	// instrument type
	g_instruIDs :ARRAY[1..g_instruTypesNum] OF INT :=[7, 8, 9, 10, 11, 12, 13, 14, 15, 16, 17, 20, 42, 43];
	
	// instrument name
	g_instruNullName :STRING := 'NULL';
	g_instruTotalLife : ARRAY[1..g_instruTypesNum] OF UINT := [11(20),100,1,1];
	g_instruNameString:ARRAY[1..g_instruTypesNum] OF STRING:=['Cadiere Forceps','Large Needle Driver','Mega SutureCut Needle Driver','Large SutureCut Needle Driver',	
															'RoundTip Scissors','Prograsp',	'Maryland Bipolar Forceps','Fenestrated Bipolar Forceps', 'Monopolar Curved Scissors',
															'Permanent Cautery Hook','Permanent Cautery Spatula','Camera','Ultrasonic Scalpel 45cm','Ultrasonic Scalpel 55cm'];
	//instrument chinese name
	g_instruNameStringCH:ARRAY[1..g_instruTypesNum] OF WSTRING:=["无创抓钳","持针钳","大号带剪刀持针钳","带剪刀持针钳","圆头直剪","细齿无创抓钳",
															"双极弧形电凝钳","双极鸭嘴电凝钳","单极弧剪","单极电钩", "单极电铲","内窥镜","超声刀 46cm","超声刀 55cm"];
	// instrument kinematic
	g_instruRodLength :ARRAY[1..g_instruTypesNum] OF LREAL :=[	0.5438,0.5438,0.5438,0.5438,	 0.5438,0.5438,0.5438, 0.5438,0.5438,	0.5432, 0.5432,0.49,0.46463,0.55225];
	g_instruHeadLength :ARRAY[1..g_instruTypesNum] OF LREAL :=[ 0.0089,0.0089,0.010,0.010,		 0.0089,0.01065,0.01065,0.01065,0.0091,	0.00935,0.00935, 0, 0, 0];
	g_instruFingerLength :ARRAY[1..g_instruTypesNum] OF LREAL :=[0.01950, 0.0096, 0.0109, 0.011, 0.01102, 0.02313, 0.019473, 0.0207, 0.01293, 0.01638, 0.01905, 0, 0, 0];

	k13:ARRAY[1..g_instruTypesNum] OF LREAL:=[0.775510204, 0.808510638, 0.590163934, 0.590163934,  0.791666667,  0.496732026, 0.590163934, 0.590163934, 0.75,   -0.663636364,	-0.663636364,   1, 1, 1];
	k23:ARRAY[1..g_instruTypesNum] OF LREAL:=[0.775510204,0.808510638, 0.590163934, 0.590163934,  0.791666667, 0.496732026, 0.590163934, 0.590163934,  0.75,   -0.663636364,	-0.663636364,   1, 1, 1];
	kx:ARRAY[1..g_instruTypesNum] OF LREAL:=[g_instruTypesNum(-1)];
	ky:ARRAY[1..g_instruTypesNum] OF LREAL:=[0.947368421, 0.947368421,0.947368421, 0.947368421, 0.947368421, 0.947368421, 0.947368421, 0.947368421, 0.947368421, 0.877192982, 0.877192982, 1, 1, 1];
	kz:ARRAY[1..g_instruTypesNum] OF LREAL:=[0.859649123, 0.824561404, 1.070175439, 1.070175439, 0.842105263, 1.342105263, 1.070175439, 1.070175439, 0.842105263, 0.964912281, 0.964912281, 1, 1, 1];
	
	g_instruMaxGripAngle:ARRAY[1..g_instruTypesNum] OF LREAL:=[45*g_deg2Rad, 40*g_deg2Rad, 40*g_deg2Rad, 40*g_deg2Rad, 40*g_deg2Rad, PI/2, 55*g_deg2Rad, 55*g_deg2Rad, PI/3, PI/6, PI/6,0,PI/4,PI/4];
	
	g_instruMaxRollAngle:ARRAY[1..g_instruTypesNum] OF LREAL:=[12(5.5), 2(g_largeNum)];
	g_instruMaxPitchAngle:ARRAY[1..g_instruTypesNum] OF LREAL:=[11(75*g_deg2Rad), 3(1)];
	g_instruMaxYawAngle:ARRAY[1..g_instruTypesNum] OF LREAL:=[9(PI/2), 90*g_deg2Rad, 90*g_deg2Rad, 3(1)];
	

	// master gripper angle limit
	g_maxMasterGripAngle :LREAL := 30*g_deg2Rad;
	g_minMasterGripAngle : LREAL :=0.0;
	g_masterGripForceStartAng :LREAL :=5*g_deg2Rad;
	
	//ultrasound knife kinematics parameter
	g_uknifeGripTravel :LREAL:= 0.00353;
	g_uknifeGripDividAngle : LREAL := 17 * g_deg2Rad;
	g_uknifeMotorLead : LREAL := 0.025;
	g_uknifeLeverRatio : LREAL := 13.0/18.5;
	
	// instrument backslash
	g_instruYawBacklash :ARRAY[1..g_instruTypesNum] OF LREAL :=[4.0*g_deg2rad, 4.0*g_deg2rad, 4.0*g_deg2rad, 4.0*g_deg2rad, 4.0*g_deg2rad, 4.0*g_deg2rad, 4.0*g_deg2rad, 4.0*g_deg2rad, 4.0*g_deg2rad,  8.0*g_deg2rad,  8.0*g_deg2rad,  0 , 0,  0 ];
	g_instruPitchBacklash :ARRAY[1..g_instruTypesNum] OF LREAL :=[3.0*g_deg2rad, 3.0*g_deg2rad, 3.0*g_deg2rad, 3.0*g_deg2rad, 3.0*g_deg2rad, 3.0*g_deg2rad, 3.0*g_deg2rad, 3.0*g_deg2rad, 3.0*g_deg2rad,  3.0*g_deg2rad,  3*g_deg2rad,  0 , 0,  0 ];
	g_instruBacklashDir: ARRAY[1..g_instruTypesNum] OF INT :=[-1, -1, -1, 0, 0];
	g_gripperCloseAng :LREAL := 2.0*g_deg2rad;
	
	// instrument grip yaw compensation
	g_instruGripYawCompAng :ARRAY[1..4] OF LREAL := [ 2*g_deg2rad,  4*g_deg2rad,  6*g_deg2rad,  8*g_deg2rad];
	g_instruGripYawCompForceLevel  :ARRAY[1..4] OF INT := [ 20, 40, 70, 101];
	
END_VAR

// ---- GVLs/GVL_interactUI.TcGVL
{attribute 'qualified_only'}
VAR_GLOBAL
	//read from UI
	//surgical status: true surgical start   false surgical finshed
	g_surgicalStatus : BOOL;

	//surgical site selection
	g_surgicalSite : UINT;

	//surgical location selection
	g_surgicalLocation : UINT;

	//stand column height limit : design 1805mm - 2495mm 
	g_heightLimit : UINT;
	g_heightLimitFromUI : UINT;
	g_heightLimitEnbale : BOOL;
	
	//ui control button enable
	g_uiCtrl : ST_uiControl;

	//ui send reset fault
	g_uiFaultReset : UINT;

	//write UI 
	//error code ID
	g_errIdType3 : UDINT;
	g_errIdType2 : UDINT;
	g_errIdType1 : UDINT;
	g_errIdType0 : UDINT;
	
	//instrument information
	g_instruInformatiom :ARRAY[1..4] OF  ST_instruInfomation;
	
	//UPS power supply mode : line voltage supply : 1 , battery powered : 2
	g_powerSupplyModeUPS : UINT;
	
	//UPS dump energy
	g_dumpEnergyUPS : UINT:=51;
	
	//ui shutdown button enable
	g_uiPowerOffEnable : BOOL;
	
	//plc confirm shutdown
	g_plcPowerOffEnable : BOOL:=FALSE;
	
	//joystick enable tip : true trigger
	g_joystickEnableTip : BOOL;
	
	//stop button signal : 0 press  , 1 No press
	g_stopButtonFormUI : UINT:=1;

	//PLC  version
	g_plcVersion : STRING := g_SWVersion;

	//Surgical guidance
	g_cartOperation : ST_cartOperation;
	
	//robot state  machine
	g_armStateMachine : ST_robotStateMachine;
	
	//scope gravity angle
	g_scopeGravityAngle : REAL;
	
	//scope type
	g_scopeType : INT;

	//fault tone current error type : 0 No fault , 1 low-level , 2 medium-level , 3 height-level
	g_curErrType : UINT;
	
	//30° endoscope face up or face down
	g_scopeUpDown : UINT := 1;
	
	//joystick signal  read RS232 data from UI
	g_joystickSignalArray : ARRAY[0..21] OF USINT;
	
	//joystick trigger
	g_joysticksTrigger : BOOL;
	
	//0: init status 1: checking 2:check succeed 3: check failed
	g_slaveSelfCheckStatus : UINT; 
	g_salveSelfCheckEnable : BOOL;
	
	//arm in disable status : 0 No disable , 1-4 number  corresponds to arms 1-4
	g_armIsDisable : UINT:=0;
	
	//the patient side has recover error flag
	g_slaveRecoverErrFlag : INT;

	//the patient side runs separately
	g_slaveRunAlone : BOOL;

	//trocar status : 0 No trocar , 1 have trocar
	g_trocarStatus : BOOL;

	//heartbeat signal
	g_heartBeat : INT;
	
	//left-right eye switch、0Left eye , 1 right eye
	g_switchLeftRightEye : INT;
	
	//the pop-up fault code is displayed
	g_popupErrorArm1 : ARRAY [0..2] OF UDINT;
	g_popupErrorArm2 : ARRAY [0..2] OF UDINT;
	g_popupErrorArm3 : ARRAY [0..2] OF UDINT;
	g_popupErrorArm4 : ARRAY [0..2] OF UDINT;
	g_popupRefresh : ARRAY [1..4] OF UINT;
	
	//instrument out of sight
	g_instruOutScope : ARRAY [1..4] OF BOOL;
	
	//arm is adjustment
	g_armIsAdjustment : ARRAY [1..4] OF UINT;
	
	//instrument max used record
	g_InstruSeriesRecord:ARRAY [1..100] OF ULINT;
END_VAR

// ---- GVLs/GVL_SafetyLogData.TcGVL
//{attribute 'qualified_only'}
VAR_GLOBAL CONSTANT
	g_maxNum:INT:=5;
	g_maxArmNum:INT:=4;
	g_maxArmJoint:INT:=13; g_maxCartJoint:INT:=8;
	g_cartNum:UDINT:=5;
	MAX_CSV_ROWS 			: UDINT := 10000;(*最大行数(任务周期为20ms)即10分钟的buffer*)
	MAX_CSV_COLUMNS 		: UDINT := 130;(*最大列数*)
	MAX_CSV_FIELD_LENGTH	: UDINT := 35;(*每个字段的字符长度*)
	MAX_CSV_RING_BUFFER		: UDINT := 5;
	g_JointNetPort:ARRAY[1..g_maxArmJoint] OF UINT :=[
		1002,    1002,	1003,	1004,	1004,	1005,	1006,	1007,	2(1008),	3(1009)];
END_VAR

VAR_GLOBAL
	g_arrayErrCodeArm:ARRAY [1..g_maxNum] OF ARRAY [0..100] OF UDINT;	
END_VAR

// ---- GVLs/GVL_SafetyParameters.TcGVL
//{attribute 'qualified_only'}
{attribute 'global_init_slot' := '49991'}
VAR_GLOBAL CONSTANT
	// safety error counts threshold to trigger fault
	g_faultTriggerCounts :INT :=10;
	
	// arm joint safety error
	g_armMaxJntEncErr :vec13d:=[g_largeNum, g_largeNum, 0.010, 4(3*g_deg2Rad), 0.010, 5(10*g_deg2Rad)];
	g_armMaxJntFollowErr :vec13d:=[g_largeNum, g_largeNum, 0.010, 4(5*g_deg2Rad), 0.010, 5(170*g_deg2Rad)];
	
	//arm joint link encoder maximum and minimum values
	g_maxLinkEnc : vec13di:=[16777215, 2(67108863), 10(16777215)];
	g_minLinkEnc : vec13di:=[13(0)];
	
	//drive error word
	g_driveErrWord : UDINT:=32;
	
	// arm joint safety error
	g_safetyJntVel : vec13d:=[2(g_largeNum), 1.0, pi, pi, pi, pi, 0.6, 5(4*pi)];
	
	// joint limit buffer(outside of joint limit)
	g_armJntPosLimitBuffer :vec13d:=[10.0*g_deg2Rad,2(0.05),4(10.0*g_deg2Rad), 0.05, 5(0)];
	
	// joint position limit
	g_minJntPos: ARRAY[1..g_sArmNum,  1..13] OF LREAL:=[(-140-50)*g_deg2Rad, 0.779-0.36, 0.00,  -1.2351,  -1.6, -170*g_deg2Rad,	-1.5-pi/2,	0.23, 5(-g_largeNum),
														(-115-50)*g_deg2Rad, 0.607-0.36, 0.00,  -1.2351,  -1.6, -170*g_deg2Rad,	-1.5-pi/2,	0.23, 5(-g_largeNum),
														(-65-50)*g_deg2Rad,  0.607-0.36, 0.00,  -1.2351,  -1.6, -170*g_deg2Rad,	-1.5-pi/2,	0.23, 5(-g_largeNum),
														(-40-50)*g_deg2Rad,  0.779-0.36, 0.00,  -1.2351,  -1.6, -170*g_deg2Rad,	-1.5-pi/2,	0.23, 5(-g_largeNum)];	
	g_maxJntPos: ARRAY[1..g_sArmNum,  1..13] OF LREAL:=[(-140+50)*g_deg2Rad, 0.779,      0.200, 4.5579,    1.6,  170*g_deg2Rad,	1.5-pi/2, 	0.58, 5(g_largeNum),
														(-115+50)*g_deg2Rad, 0.607,      0.200, 4.5579,    1.6,  170*g_deg2Rad,	1.5-pi/2, 	0.58, 5(g_largeNum),
														(-65+50)*g_deg2Rad,  0.607,      0.200, 4.5579,    1.6,  170*g_deg2Rad,	1.5-pi/2, 	0.58, 5(g_largeNum),
														(-40+50)*g_deg2Rad,  0.779,      0.200, 4.5579,    1.6,  170*g_deg2Rad,	1.5-pi/2, 	0.58, 5(g_largeNum)];	
	
	//arm joint max current
	g_maxJntCurrent : vec13d:=[2(g_largeNum),8400,7600,8400,      8400,8400,      1500,300,300,300,300, 300];
	
	// rcp position deviation for safety check
	g_rcpDeviationThres :LREAL := 0.005;
	
	//max joint commend  saltation
	g_maxJntCmdSalta : vec13d:=[2(g_largeNum), 0.010, 5(5*g_deg2Rad), 5(35*g_deg2Rad)];
	
	//max joint encoder current  saltation
	g_maxJntCurSalta : vec13d:=[2(g_largeNum), 11(60000)];
	
	// setup joint limit buffer(outside of joint limit)
	g_setupJntPosLimitBuffer :Vec5d := [5.0*g_deg2Rad, 0.01, 0.01,  2(5.0*g_deg2Rad)];
	
	// slave arm cartesion control safety error 
	g_maxCartPoseErr :ARRAY [1..6] OF LREAL:=[0.010,0.010,0.010,90*g_deg2Rad,90*g_deg2Rad,90*g_deg2Rad];
	
	//instrument open angle maximum and minimum values
	g_maxInstruOpen:LREAL;
	g_minInstruOpen:LREAL;
	
	g_motPhieErrLimit:DINT:=20000;
	
	//motor deviation between command current and feedback current limit
	g_jntCurrentCtrlLimit : vec13d:=[2(g_largeNum), 1680, 1140, 3(1680), 200, 5(g_largeNum)];
	
	// cart joint safety check limit
	g_cartMaxJntEncErr :Vec8d:=[0.01,0.01,3*g_deg2Rad,3*g_deg2Rad,0.01,3*g_deg2Rad,0.01,3*g_deg2Rad];
	g_cartMaxJntFollowErr :Vec8d:=[0.01,0.01,3*g_deg2Rad,3*g_deg2Rad,0.01,3*g_deg2Rad,0.01,3*g_deg2Rad];
	g_cartMaxLinkEnc :Vec8di:=[4(1), 67108863,16777215,67108863,16777215] ;
	g_cartMinLinkEnc :Vec8di:=[4(1),  4(0)];
	g_cartMaxJntVel :Vec8d:=[0.0025*2,0.0025*2,2.3*2,2.3*2, 0.080, 10*g_deg2Rad, 0.10, 10*g_deg2Rad];
	g_cartMaxJntCurrent :Vec8d:=[1080*2,1080*2,19800*2,19800*2, 10000*2,3800*2,3800*2,3800*2];
	g_cartMinJntPos :Vec8d:=[0,		0,		1, 1,  0-0.01,		-35*g_deg2Rad,	0-0.02,		-165*g_deg2Rad];
	g_cartMaxJntPos :Vec8d:=[0.053,0.053,1, 1,  0.69+0.01, 35*g_deg2Rad,	0.5+0.02,	165*g_deg2Rad];
END_VAR

// ---- GVLs/GVL_SystemParameters.TcGVL
VAR_GLOBAL CONSTANT
		
	g_SWVersion : STRING := '2(1.0.0.1)';
	
	g_mArmNum :INT := 2;	
	g_mJntNum :INT := 7;	
	g_sArmNum :INT := 4;	
	g_sJntNum :INT := 8;
	g_setupJntNum :INT :=5;
	g_cartDofs :INT :=6;
	g_cartJntNum:INT :=8;
	
	
	
	// control loop interval for each task
	g_slaveArmCtrlCycleTime :LREAL :=0.00025;
	g_slaveArmCtrlFreq :LREAL :=1.0/g_slaveArmCtrlCycleTime;
	g_armDynamicCycleTime :LREAL := 0.001;
	g_armDynamicFreq :LREAL := 1.0/g_armDynamicCycleTime;
	g_setupArmCtrlCycleTime :LREAL := 0.001;
	g_setupArmCtrlFreq :LREAL := 1.0/g_setupArmCtrlCycleTime;
	g_cartCtrlCycleTime :LREAL := 0.001;
	g_cartCtrlFreq :LREAL := 1.0/g_cartCtrlCycleTime;
	
	// wait time before robot init  for ethercat to stablize 
	g_robotInitWaitTime : LREAL := 5.0;

	g_robotSafetyCheckWaitTime : LREAL :=6.0;
END_VAR

// ---- GVLs/SetupArms/GVL_SetupJointEncoderCaliData.TcGVL
{attribute 'qualified_only'}
// Robot8 --joints parameters of setup arms
VAR_GLOBAL
	// absolute encoder value at minimal joint positon
	g_minLinkEncoder :ARRAY[1..g_sArmNum, 1..g_setupJntNum] OF DINT :=
		[123569, 35609025, 57736, 7242080, 8849999,
		 76588 , 33880077, 23270, 11506200, 2528900,
		  92809, 39087738, 30100, 90344, 45244,
		  97353, 37341559, 26764, 2969850, 13989400];
		 
	// absolute encoder value at maximum joint positon
	g_maxLinkEncoder :ARRAY[1..g_sArmNum, 1..g_setupJntNum] OF DINT :=
		[29697 , 34190666, 1678, 5374722, 468900,
		 113660, 32457000, 31924, 9643400, 10948070,
		 129919 , 37687900,  39566, 104908, 111011,
		  4419 , 35927748, 36194, 1105500, 5653000];
	
	// absolute encoder value at calibrated positon
	g_caliLinkEncoder :ARRAY[1..g_sArmNum, 1..g_setupJntNum] OF DINT :=
		[10043, 34190666, 57736, 14420666, 13062300,
		  94700, 32457000, 23270, 1922210, 6757000,
		 111618, 37687900, 30100 , 35294, 78076,
		  117777, 35927748, 26764, 10044500, 1409000];
	
	 // if absolute encoder value cross zeros within joint motion range
	g_linkEncZeroCross :ARRAY[1..g_sArmNum, 1..g_setupJntNum] OF INT :=
		[1, 0, 1, 1, 1,
		 0, 0, 0, 1, 0,
		 0, 0, 0, 1, 0,
		 1, 0, 0, 1, 1];
		 
//################ DO NOT modify parameters below ###########################
	// abolute encoder expanded limit buffer in case there is calibrtion error at limit position
    g_linkEncLimitBuffer : ARRAY [1..g_setupJntNum] OF DINT := [2000, 100000, 100, 2(100000)];
	g_linkEncLimitBufferFR : ARRAY [1..g_setupJntNum] OF DINT := [2(2000),100, 2(2000)];

	// absolute encoder direction
	g_asbEncoderDir :ARRAY[1..g_setupJntNum] OF INT :=[1, -1, 1, 1, -1];
	g_asbEncoderDirFR :ARRAY[1..g_setupJntNum] OF INT :=[1, -1, 1, -1, 1];
													
	// flag if joint can rotate multiple cycles
	g_multipleCyclesJoint :ARRAY[1..g_sArmNum, 1..g_setupJntNum] OF INT :=
		[0, 0, 0, 0, 0,
		 0, 0, 0, 0, 0,
		 0, 0, 0, 0, 0,
		 0, 0, 0, 0, 0];
		 
	// joint position at link encoder calibrated point
	g_linkEncCaliJntPos :ARRAY[1..g_sArmNum, 1..g_setupJntNum] OF LREAL :=
		[-140*g_deg2Rad, 0.779, 0.0, 90.0*g_deg2Rad, 0.0,
		 -115*g_deg2Rad, 0.607, 0.0, 90.0*g_deg2Rad, 0.0,
		 -65*g_deg2Rad, 0.607, 0.0, 90.0*g_deg2Rad, 0.0,
 		 -40*g_deg2Rad, 0.779, 0.0, 90.0*g_deg2Rad, 0.0];
	
END_VAR

// ---- GVLs/SetupArms/GVL_SetupMotorParameters.TcGVL
{attribute 'global_init_slot' := '49991'}
{attribute 'qualified_only'}
VAR_GLOBAL CONSTANT
	// encoder resolution
	//TODO: resolution of joint 2/3 need verification
	g_incEncoderRes :ARRAY[1..g_setupJntNum] OF DINT :=[5(65536)];
	g_absEncoderRes :ARRAY[1..g_setupJntNum] OF DINT :=[131072,8192, 65536, 2(16777215)];
	g_absEncoderResFR :ARRAY[1..g_setupJntNum] OF DINT :=[131072,8192, 65536, 2(131072)];
	
	// reduction ratio
	g_motorReduction :ARRAY[1..g_setupJntNum] OF LREAL :=[1,1,2*pi/0.1256,81,160];
	g_absEncoderReduction :ARRAY[1..g_setupJntNum] OF LREAL :=[1.0, 2*pi/0.002 , 2*PI/(0.09995*16), 1.0, 1.0];
	
	// motor parameters
	g_motorTrqConst :ARRAY[1..g_setupJntNum] OF LREAL :=[ 1,1,1.35/5.3,0.38/3.8,0.9/5.6];
	g_motorMaxCurrent :ARRAY[1..g_setupJntNum] OF LREAL :=[ 1,1,8000,3800,5600];//mA
	
	// motor and absEncoder direction
	g_motorDir :ARRAY[1..g_setupJntNum] OF INT :=[-1, -1, -1, -1, 1];
																												 
	// joint position limit
	g_minJntPos: ARRAY[1..g_sArmNum,  1..g_setupJntNum] OF LREAL:=[ (-140-50)*g_deg2Rad, 0.779-0.36,0.00,-1.2351,-1.6,
																	(-115-50)*g_deg2Rad, 0.607-0.36,0.00,-1.2351,-1.6,
																	(-65-50)*g_deg2Rad, 0.607-0.36,0.00,-1.2351,-1.6,
																	(-40-50)*g_deg2Rad, 0.779-0.36,0.00,-1.2351,-1.6];	
	g_maxJntPos: ARRAY[1..g_sArmNum,  1..g_setupJntNum] OF LREAL:=[ (-140+50)*g_deg2Rad, 0.779,0.200,4.5579,1.6,
																	(-115+50)*g_deg2Rad, 0.607,0.200,4.5579,1.6,
																	(-65+50)*g_deg2Rad, 0.607,0.200,4.5579,1.6,
																	(-40+50)*g_deg2Rad, 0.779,0.200,4.5579,1.6];	
	
	// joint velocity limit
	g_maxJntVel :ARRAY[1..g_setupJntNum] OF LREAL :=[0.1, 0.1, 0.1, 0.1, 0.1];
	
END_VAR

// ---- GVLs/SlaveArms/GVL_SlaveControlParameters.TcGVL
{attribute 'global_init_slot' := '49991'}
VAR_GLOBAL CONSTANT
	// slave arm joint position controller parameters
	g_posKp :ARRAY[1..g_sJntNum] OF LREAL :=[2000.0, 2000.0, 10000.0, 5(5)];
	g_posKd :ARRAY[1..g_sJntNum] OF LREAL :=[200.0, 200.0, 1000.0, 5(0.25)];
	g_posKi :ARRAY[1..g_sJntNum] OF LREAL :=[2000.0, 2000.0, 10000.0, 5(10.0)];
	g_posKiLimit :ARRAY[1..g_sJntNum] OF LREAL :=[2500,2500,  500, 5(75)];// define in current
	g_posCtrlLimit :ARRAY[1..g_sJntNum] OF LREAL :=[5600,5600,  1300, 5(200)];// define in current
	
	// control tolerance
	g_jntCtrlAngTolLow :LREAL :=0.2*g_deg2Rad;
	g_jntCtrlAngTolHigh :LREAL :=2*g_deg2Rad;
	g_cartCtrlPosTolLow :LREAL :=0.0002;
	g_cartCtrlOriTolLow :LREAL :=0.2*g_deg2Rad;
	g_cartCtrlPosTolHigh :LREAL :=0.001;
	g_cartCtrlOriTolHigh :LREAL :=2*g_deg2Rad;
	
	// filter cut-off frequency for velocity and torque
	g_curJntVelLpfCutoffFreq :LREAL := 30;
	g_cmdJntTrqLpfCutoffFreq :LREAL := 300;
	g_curJntTrqLpfCutoffFreq :LREAL := 300;
		
	// controller would keep command unchanged when error 
	// between command and current value is less than this value
	g_jntCtrlErrForCmdHold :LREAL :=1.0*g_deg2Rad;
	
	// joint is assumed to be static if velocity is less than this value
	g_jntStaticVelThres :LREAL :=0.2*g_deg2Rad;
	
	// joint velocity threshold for full friction compensation
	g_fullFrictionVel :LREAL :=2.0*g_deg2Rad;
	
	// friciton compensation scael
	g_frictionCompScale :LREAL := 0.8;
	
END_VAR

// ---- GVLs/SlaveArms/GVL_SlaveJointEncoderCaliData.TcGVL
{attribute 'qualified_only'}
// Robot8 --joints parameters of slave arms
VAR_GLOBAL CONSTANT	
	// absolute encoder value at minimal joint positon
	g_minLinkEncoder :ARRAY[1..g_sArmNum, 1..g_sJntNum] OF DINT :=
		[15026800, 7686890, 24511, 0, 0, 0, 0, 0,
		 10489100, 4588800, 10330, 0, 0, 0, 0, 0,
		35  , 85624, 57700, 0, 0, 0, 0, 0,
		 6116900,  5078766,61396 , 0, 0, 0, 0, 0];
		 
	// absolute encoder value at maximum joint positon
	g_maxLinkEncoder :ARRAY[1..g_sArmNum, 1..g_sJntNum] OF DINT :=
		[13899866 , 276216, 46808, 0, 0, 0, 0, 0,
		 9367400, 12196650, 53080 , 0, 0, 0, 0, 0,
		  8803  , 14040, 14555, 0, 0, 0, 0, 0,
		 4991310,  12616170,18239, 0, 0, 0, 0, 0];
	
	// absolute encoder value at calibrated positon
	g_caliLinkEncoder :ARRAY[1..g_sArmNum, 1..g_sJntNum] OF DINT :=
		[6048200, 4849470, 46808, 46180 , 6018 , 49928 , 23680 , 34680, 
		 1548800, 9172500, 10330, 57272 , 13688 , 48750 , 43310 , 13951 ,
		  69906, 107792, 14555, 17188 , 38930,  40400,  35192, 5020 ,
		 13906777,  9940888, 18192 , 45120,  52590,  52590,  64913,  38950];
	
	 // if absolute encoder value cross zeros within joint motion range
	 // NOTICE: joint 7 is always 0.
	g_linkEncZeroCross :ARRAY[1..g_sArmNum, 1..g_sJntNum] OF INT :=
		[1, 0, 1, 1, 1, 1, 1, 1,
		 1, 0, 0, 1, 1, 1, 1, 1,
		 1, 1, 0, 1, 1, 1, 1, 1,
		 1, 0, 0, 1, 1, 1, 1, 1];
		 
	 // joint SDO address
	g_slaveArmNetID: ARRAY[1..4] OF T_AmsNetId:=['169.254.223.120.10.1','192.168.2.91.4.1','192.168.2.91.6.1','192.168.2.91.5.1'];
	g_slaveJointNetPort:ARRAY[1..g_sArmNum,1..g_sJntNum] OF UINT :=[
		1005,	1006,	1007,	2(1008),	3(1009),
		1005,	1006,	1007,	2(1008),	3(1009),
		1005,	1006,	1007,	2(1008),	3(1009),
		1005,	1006,	1007,	2(1008),	3(1009)];
		
//################ DO NOT modify parameters below ###########################
	// abolute encoder expanded limit buffer in case there is calibrtion error at limit position
	g_linkEncLimitBuffer :ARRAY [1..g_sJntNum] OF DINT := [2(100000),6(1000)];
	g_linkEncLimitBufferFR :ARRAY [1..g_sJntNum] OF DINT := [2(1000),6(1000)];
	
	// absolute encoder direction
	g_asbEncoderDir :ARRAY[1..g_sJntNum] OF INT :=[1, -1, -1, -1, -1, -1, -1, -1];
	g_asbEncoderDirFR :ARRAY[1..g_sJntNum] OF INT :=[-1, 1, -1, -1, -1, -1, -1, -1];
	
	// flag if joint can rotate multiple cycles
	g_multipleCyclesJoint :ARRAY[1..g_sArmNum, 1..g_sJntNum] OF INT :=
		[0, 0, 0, 1, 1, 1, 1, 1,
		 0, 0, 0, 1, 1, 1, 1, 1,
		 0, 0, 0, 1, 1, 1, 1, 1,
		 0, 0, 0, 1, 1, 1, 1, 1];
		 
	// joint position at link encoder calibrated point
	g_linkEncCaliJntPos :ARRAY[1..g_sJntNum] OF LREAL :=
		[0.0, -111.22*pi/180, 0.54608, 5(0.0)];

	
END_VAR

// ---- GVLs/SlaveArms/GVL_SlaveMotorParameters.TcGVL
{attribute 'global_init_slot' := '49991'}
{attribute 'qualified_only'}
VAR_GLOBAL CONSTANT
	// encoder resolution
	g_incEncoderRes :ARRAY[1..g_sJntNum] OF DINT :=[2(65536),4096,5(65536)];
	g_absEncoderRes :ARRAY[1..g_sJntNum] OF DINT :=[2(16777216),6(65536)];
	g_absEncoderResFR :ARRAY[1..g_sJntNum] OF DINT :=[2(131072),6(65536)];
	
	// reduction ratio
	g_motorReduction :ARRAY[1..g_sJntNum] OF LREAL :=[ 81,81,  2*pi/0.006, 5(388125.0/4693)];
	g_absEncoderReduction :ARRAY[1..g_sJntNum] OF LREAL :=[2(1.0), 2*PI/0.486, 5(1.0)];
	
	// motor parameters
	g_motorTrqConst :ARRAY[1..g_sJntNum] OF LREAL :=[ 0.9/5.6,0.9/5.6, 0.032,5(0.0193)];
	g_motorMaxCurrent :ARRAY[1..g_sJntNum] OF LREAL :=[ 5600,5600,  1300, 5(250)];//mA
	
	// motor encoder direction
	g_motorDir :ARRAY[1..g_sJntNum] OF INT :=[-1, 1, -1, 1, 1, 1, 1, 1];
																 
	// joint position limit
	g_minJntPos: ARRAY[1..g_sJntNum] OF LREAL:=[-2.7,	-1.5-pi/2,	0.23, 	5(-g_largeNum)];	
	g_maxJntPos: ARRAY[1..g_sJntNum] OF LREAL:=[2.7,		1.13-pi/2, 	0.58, 	5(g_largeNum)];
	
	// DH joint position limit
	//NOTE: wrist pitch and yaw angle is reset after instrument is mounted 
	g_minDHJntPos : ARRAY[1..6] OF LREAL :=[-2.7,	-1.5-pi/2,	0.235, -5.5, -PI/2 - 75*g_deg2Rad , -PI/2];
	g_maxDHJntPos : ARRAY[1..6] OF LREAL :=[2.7,	1.13-pi/2, 	0.535, 5.5, -PI/2 + 75*g_deg2Rad, PI/2];
	
	// joint velocity limit
	g_maxJntVel :ARRAY[1..g_sJntNum] OF LREAL :=[1.25, 1.25, 0.5, 5(7.0)];
		
END_VAR

// ---- FBs_Robots/FB_Instrument.TcPOU
FUNCTION_BLOCK FB_Instrument

VAR_IN_OUT CONSTANT
	i_slaveArm	:FB_SlaveArm;
END_VAR

VAR
	// instrument type
	m_instruType : 	E_InstrumentType := InstruType_UNKNOWM;
	
	// instrument name
	m_instruName : STRING:= g_instruNullName;
	m_instruNameCH : WSTRING;
	
	// instrument type index, which is used to get relative parameters from global variable arrays
	m_instruTypeIdx :INT:=0;
	
	// flag if instrument is singer finger
	m_isSingleFinger:BOOL:= FALSE;
	
	//flag if instrument is energy type 
	m_isEnergyType : UINT :=0;
	
	// current and max allowed read tries
	m_curReadTries :INT :=0;
	m_maxReadTries :INT := 2;
	
	//IP of operating arm
	m_armNetId:T_AmsNetId; 	
	
	//Joint port number
	m_jointInstruAddr:UINT;	

	//Arm LED Prot	
	m_LEDPortAddr:UINT;		
	
	//The state and parameters readed from the instrument
	m_onChipData:ST_InstruOnChipData;
	
	// instrument kinematic parameters
	m_kinematicParameters:ST_InstruKinematicParam; 
	
	// joint position when instrument is at ZERO posture
	m_jntPosOffset:Vec8d;
	
	// reduction from motor joint to endoscope rotate joint
	m_endoscopeRotateReduction :LREAL := 2.0/3.0;
	
	//endoscope type
	m_curEndoscopeType :E_EndoscopeType:=EndoScopeType_30;
	m_nextEndoscopeType :E_EndoscopeType:=EndoScopeType_30;
	
	//endoscope posutre
	m_curEndoscopePosture :E_EndoscopePosture:=EndoscopePosture_HeadDown;
	m_nextEndoscopePosture :E_EndoscopePosture:=EndoscopePosture_HeadDown;
	
	// udint code for zero position
	m_zeroPosCode : UDINT;
	
	// joint4 zero position, which is supposed to be a contant value
	m_jnt4ZeroPos :LREAL := 5.7;
	
	//reset arm  LED flag
	m_resetArmLEDFlag : BOOL :=TRUE;
	
	// variables used to read instrument information
	m_Step:INT;
	m_Value:UDINT;
	m_ReadDelay:TON;
	m_DealyTime:TIME:=T#0.5S;
	m_IDReadResult:UDINT;
	m_IDResult:ULINT;
	m_SeriesReadResult:UDINT;
	m_PosReadResult:UDINT;
	m_PosL1,m_PosL2,m_PosL3:UDINT;
	m_signL1,m_signL2,m_signL3:UDINT;
	m_UsageReadResult:ULINT;
	m_InstruUsageToLED:ULINT;
	m_InstruSeriesRecord:ARRAY [1..100] OF ULINT;
	m_HaveRecord:BOOL;
	m_SdoWrite:FB_EcCoESdoWrite;
	m_SdoRead:FB_EcCoESdoRead;
	
	//variables used to read-write instrument number of use
	m_useNumStep : INT;
	m_ReadNumDelay:TON;
	m_useNumReadResult:ULINT;
	m_useNumSendToLED:ULINT;
	
	// rising edge generator for instrument information reading
	m_writeLDP:R_TRIG;
	
END_VAR

METHOD PROTECTED checkInstruType : BOOL
VAR_INPUT
END_VAR
VAR
	i:INT;
END_VAR
// search instrument type
m_instruTypeIdx:=0;
FOR i:=1 TO g_instruTypesNum DO
	IF g_instruIDs[i] = m_onChipData.m_InstruID THEN
		m_instruTypeIdx := i;
		EXIT;
	END_IF
END_FOR

// return directly if instrument ID is invalid
checkInstruType := m_instruTypeIdx >0;
IF NOT(checkInstruType) THEN
	RETURN;
END_IF

// instrument type and name
m_instruType := m_onChipData.m_InstruID;
m_instruName :=GVL_InstruCtrlParams.g_instruNameString[m_instruTypeIdx];
m_instruNameCH := GVL_InstruCtrlParams.g_instruNameStringCH[m_instruTypeIdx];

// check if instrument has one finger
m_isSingleFinger :=  (m_instruType = InstruType_CauteryHook OR  m_instruType = InstruType_CauterySpatula );

// check the type of energy instrument
IF m_instruType = InstruType_CurvedScissors OR m_instruType = InstruType_CauteryHook OR m_instruType = InstruType_CauterySpatula THEN
	m_isEnergyType := 1;
ELSIF m_instruType = InstruType_MarylandForceps OR m_instruType = InstruType_FenestratedForceps THEN
	m_isEnergyType := 2;
ELSIF m_instruType = InstruType_UltrasoundKnifeS OR m_instruType = InstruType_UltrasoundKnifeU THEN
	m_isEnergyType := 3;
ELSE
	m_isEnergyType := 0;
END_IF


// update instrument kinematic parameters based on readed info
IF m_instruTypeIdx > 0 THEN
	m_kinematicParameters.m_maxGripAngle := g_instruMaxGripAngle[m_instruTypeIdx];
	
	m_kinematicParameters.k13:=k13[m_instruTypeIdx];
	m_kinematicParameters.k23:=k23[m_instruTypeIdx];
	m_kinematicParameters.kx:=kx[m_instruTypeIdx];
	m_kinematicParameters.ky:=ky[m_instruTypeIdx];
	m_kinematicParameters.kz:=kz[m_instruTypeIdx];
			
	m_kinematicParameters.m_rodLength := GVL_InstruCtrlParams.g_instruRodLength[m_instruTypeIdx] - GVL_SlaveArmKinematic.g_panelHeight;
	m_kinematicParameters.m_headLength := GVL_InstruCtrlParams.g_instruHeadLength[m_instruTypeIdx];
	m_kinematicParameters.m_fingerLength := GVL_InstruCtrlParams.g_instruFingerLength[m_instruTypeIdx];

	m_kinematicParameters.m_wristMinDHJntPos[1]:=-GVL_InstruCtrlParams.g_instruMaxRollAngle[m_instruTypeIdx];
	m_kinematicParameters.m_wristMaxDHJntPos[1]:=GVL_InstruCtrlParams.g_instruMaxRollAngle[m_instruTypeIdx];
	m_kinematicParameters.m_wristMinDHJntPos[2]:=-GVL_InstruCtrlParams.g_instruMaxPitchAngle[m_instruTypeIdx]-pi/2;
	m_kinematicParameters.m_wristMaxDHJntPos[2]:=GVL_InstruCtrlParams.g_instruMaxPitchAngle[m_instruTypeIdx]-pi/2;
	m_kinematicParameters.m_wristMinDHJntPos[3]:=-GVL_InstruCtrlParams.g_instruMaxYawAngle[m_instruTypeIdx];
	m_kinematicParameters.m_wristMaxDHJntPos[3]:=GVL_InstruCtrlParams.g_instruMaxYawAngle[m_instruTypeIdx];

END_IF
END_METHOD

PROPERTY curScopePosture : E_EndoscopePosture
GET
curScopePosture:= m_curEndoscopePosture;
END_GET
SET
m_curEndoscopePosture := curScopePosture;
END_SET
END_PROPERTY

PROPERTY curScopeType : E_EndoscopeType
GET
curScopeType := m_curEndoscopeType;
END_GET
SET
m_curEndoscopeType := curScopeType;
END_SET
END_PROPERTY

METHOD PUBLIC gripAngleMap : BOOL
VAR_INPUT
	// master gripper angle
	i_masterGripAng :LREAL;
END_VAR

VAR_OUTPUT
	// slave instrument gripper angle
	o_instruGripAngle :LREAL;
	
	// slave instrument grip force	
	o_instruGripForceLevel :LREAL;
END_VAR

VAR
	gripLevel :REAL;
END_VAR
// suppose finger is  closed and zero force if instrument has only one finger
IF m_isSingleFinger THEN
	o_instruGripAngle := 0;
	o_instruGripForceLevel:= 0;
	RETURN;
END_IF 

// finger closed and force applied
IF i_masterGripAng < g_masterGripForceStartAng THEN
	o_instruGripAngle := m_kinematicParameters.m_minGripAngle;
	// NOTE: force is applied from 50%，as minimum gripper angle already apply some sort of force
	o_instruGripForceLevel := 50+50*(g_masterGripForceStartAng - i_masterGripAng)/(g_masterGripForceStartAng - g_minMasterGripAngle);
// finger open
ELSE
	o_instruGripAngle := (g_maxMasterGripAngle - i_masterGripAng)/(g_maxMasterGripAngle - g_masterGripForceStartAng);
	o_instruGripAngle :=m_kinematicParameters.m_maxGripAngle - o_instruGripAngle * (m_kinematicParameters.m_maxGripAngle - m_kinematicParameters.m_minGripAngle);
	o_instruGripAngle := LIMIT(m_kinematicParameters.m_minGripAngle, o_instruGripAngle, m_kinematicParameters.m_maxGripAngle );
	o_instruGripForceLevel:=0;
END_IF
END_METHOD

METHOD PUBLIC init : BOOL
VAR_INPUT
	armIdx :INT;
END_VAR
VAR
	i:INT;
END_VAR
//Update the IP and port number of the operating arm
m_armNetId:=GVL_SlaveJointEncoderCaliData.g_slaveArmNetID[armIdx];
m_jointInstruAddr:=GVL_SlaveJointEncoderCaliData.g_slaveJointNetPort[armIdx,4];

// init joint motion range
FOR i:=1 TO 3 DO
	m_kinematicParameters.m_wristMinDHJntPos[i]:=GVL_SlaveMotorParameters.g_minDHJntPos[i+3];
	m_kinematicParameters.m_wristMaxDHJntPos[i]:=GVL_SlaveMotorParameters.g_maxDHJntPos[i+3];
END_FOR
END_METHOD

METHOD PUBLIC initInstruJntPos : BOOL
VAR_INPUT
	m_curJntPos :Vec8d;
END_VAR

VAR
	i:INT;
END_VAR

FOR i := 4 TO 8 BY 1 DO
	m_jntPosOffset[i]:=m_curJntPos[i];
END_FOR
END_METHOD

// convert motor joint position to DH joint position
METHOD PUBLIC instruFK : BOOL
VAR_IN_OUT CONSTANT
	// motor joint position of slave arm
	i_jntPos :Vec8d;
END_VAR

VAR_IN_OUT
	// instrument DH  joint positon
	r_DHJntPos :Vec6d;

	// gripper angle
	r_gripAngle :LREAL;
END_VAR

VAR
	jntPosL1,jntPosL2,jntPosL3,jntPosL4,jntPosL5 :LREAL;
	gripAngle:LREAL;
END_VAR
r_DHJntPos[1]:=i_jntPos[1];
r_DHJntPos[2]:=i_jntPos[2];
r_DHJntPos[3]:=i_jntPos[3];

// ################## endoscope ############################
IF m_instruType = InstruType_endoscope THEN
	r_DHJntPos[4]:=m_endoscopeRotateReduction*(i_jntPos[8]-m_jntPosOffset[8]);
	IF m_curEndoscopeType = EndoScopeType_30 THEN
		r_DHJntPos[5]:=-pi/2+30*g_deg2Rad;
	ELSE
		r_DHJntPos[5]:=-pi/2;
	END_IF
	r_DHJntPos[6]:=0;
	RETURN;
END_IF

// ################## ultrosonic knief ############################
IF m_instruType = InstruType_UltrasoundKnifeS OR m_instruType = InstruType_UltrasoundKnifeU THEN
	r_DHJntPos[4]:=-(i_jntPos[8]-m_jntPosOffset[8])/m_kinematicParameters.kx;
	r_DHJntPos[5]:=-pi/2;
	r_DHJntPos[6]:=0;
	r_gripAngle:=ultrasoundKnifeGripAngleFK(i_jntPos[6]-m_jntPosOffset[6]);
	RETURN;
END_IF


//#################### instrument forward kinematic ############
// convert motor joint position to instrument joint position
jntPosL1:=(i_jntPos[4]-m_jntPosOffset[4]);
jntPosL2:=(i_jntPos[5]-m_jntPosOffset[5]);
jntPosL3:=(i_jntPos[6]-m_jntPosOffset[6]);
jntPosL4:=-(i_jntPos[7]-m_jntPosOffset[7]);
jntPosL5:=-(i_jntPos[8]-m_jntPosOffset[8]);

// diable L1 if instrument is single finger
IF m_isSingleFinger THEN
	jntPosL1 := -jntPosL2;
END_IF

// instrument FK in local coordinate
r_DHJntPos[4]:=jntPosL4/m_kinematicParameters.kx;
r_DHJntPos[5]:=jntPosL3/m_kinematicParameters.ky;
r_DHJntPos[6]:=(jntPosL1-jntPosL2-2*r_DHJntPos[5]*m_kinematicParameters.k13*m_kinematicParameters.kz)/(2*m_kinematicParameters.m_openAngleDir*m_kinematicParameters.kz);

// convert instrument rotation to arm DH joint position
r_DHJntPos[5]:=-r_DHJntPos[5]-pi/2;
r_DHJntPos[6]:=-r_DHJntPos[6];

// grip angle
gripAngle:=(jntPosL1+jntPosL2)/(m_kinematicParameters.m_openAngleDir*m_kinematicParameters.kz);

//################### gripper angle handle #################
IF (InstruType_ProGraspForceps=m_instruType) THEN//细齿无创抓钳
	proGrsapForcepsGripAngleFK(frontAngle:= gripAngle, endAngle=> r_gripAngle);

ELSIF (InstruType_CauteryHook = m_instruType) THEN//单级电钩
	r_gripAngle:=0;
ELSE
	r_gripAngle:=gripAngle;
END_IF
END_METHOD

METHOD PROTECTED InstruIDRecord :ARRAY [1..100] OF  ULINT
VAR_INPUT
	i_NewValue:ULINT;
	i_ArrayData:ARRAY [1..100] OF ULINT;
END_VAR

VAR
	k1:INT;
	Have_Data:BOOL;
END_VAR

FOR k1:= 1 TO 100 BY 1 DO
	IF i_NewValue=i_ArrayData[k1] THEN
		Have_Data:=TRUE;
		EXIT;
	ELSE
		Have_Data:=FALSE;
	END_IF
END_FOR

IF Have_Data=FALSE THEN
	FOR k1:= 1 TO 99 BY 1 DO
		InstruIDRecord[k1+1]:=i_ArrayData[k1];
	END_FOR
	InstruIDRecord[1]:=i_NewValue;
ELSE
	InstruIDRecord:=i_ArrayData ;
END_IF
END_METHOD

METHOD PUBLIC instruIK : BOOL
VAR_INPUT
	// DH  joint positon
	i_DHJntPos :Vec6d;

	// gripper angle
	i_gripAngle :LREAL;
	
END_VAR
VAR_OUTPUT
	o_jntPos:Vec8d;
END_VAR
VAR
	gripAngle:LREAL;
	i:INT;
	rot_x:lreal;
	rot_y:lreal;
	rot_z:lreal;

	kx,ky,kz,k13,k23:LREAL;
	open_direction:INT;
	
	d,ra:LREAL;
	AngleOffsetL3:LREAL;
	m_targetOffsetL3:LREAL;
	m_actOffsetL3:LREAL;
	
	m_gripAnglePbox:Vec8d;

	L3Offset:LREAL:=-3;
END_VAR
o_jntPos[1] := i_DHJntPos[1];
o_jntPos[2] := i_DHJntPos[2];
o_jntPos[3] := i_DHJntPos[3];

// ################## endoscope ############################
IF m_instruType = InstruType_endoscope THEN
	o_jntPos[8] := i_DHJntPos[4]/m_endoscopeRotateReduction + m_jntPosOffset[8];
	o_jntPos[4]:=0;
	o_jntPos[5]:=0;
	o_jntPos[6]:=0;
	o_jntPos[7]:=0;
	RETURN;
END_IF

//################### gripper angle handle #################
IF (12=onChipData.m_InstruID) THEN//细齿无创抓钳
	proGrsapForcepsGripAngleIK(endAngle:= i_gripAngle, frontAngle=> gripAngle);
	
ELSIF 16 = onChipData.m_InstruID THEN//单级电钩\电铲
	gripAngle:=0;
	
ELSE
	gripAngle:=i_gripAngle;
END_IF

// ################# instrument inverse kinematic ##############
// convert arm DH joint position to  instrument rotation
rot_x:=i_DHJntPos[4];
rot_y:=-i_DHJntPos[5]-pi/2;
rot_z:=-i_DHJntPos[6];

// instrument IK in local coordinate
k13:=m_kinematicParameters.k13;
k23:=m_kinematicParameters.k23;
kx:=m_kinematicParameters.kx;
ky:=m_kinematicParameters.ky;
kz:=m_kinematicParameters.kz;
d:=m_kinematicParameters.m_openAngleDir;

// ################## ultrosonic knief ############################
IF InstruType_UltrasoundKnifeS = onChipData.m_InstruID OR InstruType_UltrasoundKnifeU = onChipData.m_InstruID THEN
	m_gripAnglePbox[4]:=0;
	m_gripAnglePbox[5]:=0;
	m_gripAnglePbox[6]:=ultrasoundKnifeGripAngleIK(gripAngle); 
	m_gripAnglePbox[7]:=rot_x*kx;
	m_gripAnglePbox[8]:=rot_x*kx;
ELSE
	m_gripAnglePbox[7]:=rot_x*kx;
	m_gripAnglePbox[6]:=rot_y*ky;
	ra:=gripAngle;
	m_gripAnglePbox[4]:=rot_y*k13*kz+d*rot_z*kz+d*ra*kz/2;
	m_gripAnglePbox[5]:=-rot_y*k23*kz-d*rot_z*kz+d*ra*kz/2;
END_IF

// convert instrument joint position to motor joint position
o_jntPos[4] := m_gripAnglePbox[4] + m_jntPosOffset[4];
o_jntPos[5] := m_gripAnglePbox[5] + m_jntPosOffset[5];
o_jntPos[6] := m_gripAnglePbox[6] + m_jntPosOffset[6];
o_jntPos[7] := -m_gripAnglePbox[7] + m_jntPosOffset[7];
o_jntPos[8] := -m_gripAnglePbox[8] + m_jntPosOffset[8];
END_METHOD

// convert motor joint velocity to DH joint velocity
METHOD PUBLIC instruJntVelFK : BOOL
VAR_IN_OUT CONSTANT
	// motor joint velocity of slave arm
	i_jntVel :Vec8d;
END_VAR

VAR_IN_OUT
	// instrument DH  joint velocity
	r_DHJntVel :Vec6d;
END_VAR

VAR
	jntPosL1,jntPosL2,jntPosL3,jntPosL4,jntPosL5 :LREAL;
	gripAngle:LREAL;
END_VAR
r_DHJntVel[1]:=i_jntVel[1];
r_DHJntVel[2]:=i_jntVel[2];
r_DHJntVel[3]:=i_jntVel[3];

r_DHJntVel[4]:=-i_jntVel[7]/m_kinematicParameters.kx;
r_DHJntVel[5]:=i_jntVel[6]/m_kinematicParameters.ky;
r_DHJntVel[6]:=(i_jntVel[4]-i_jntVel[5]-2*r_DHJntVel[5]*m_kinematicParameters.k13*m_kinematicParameters.kz)/(2*m_kinematicParameters.m_openAngleDir*m_kinematicParameters.kz);
r_DHJntVel[5]:=-r_DHJntVel[5];
r_DHJntVel[6]:=-r_DHJntVel[6];
END_METHOD

PROPERTY instruName : String
GET
instruName := m_instruName;
END_GET
END_PROPERTY

PROPERTY instruNameCH : WSTRING
GET
instruNameCH := m_instruNameCH;
END_GET
END_PROPERTY

METHOD PROTECTED InstruSreiesFind : BOOL
VAR_INPUT
	i_NewValue:ULINT;
	i_ArrayData:ARRAY [1..100] OF ULINT;
	
END_VAR

VAR
	k1:INT;
END_VAR
InstruSreiesFind:=FALSE;
FOR k1:= 1 TO 100 BY 1 DO
	IF i_NewValue=i_ArrayData[k1] THEN
		InstruSreiesFind:=TRUE;
		EXIT;
	ELSE
		InstruSreiesFind:=FALSE;
	END_IF
END_FOR
END_METHOD

PROPERTY PUBLIC instruType : INT
GET
instruType := m_instruType;
END_GET
END_PROPERTY

PROPERTY isEnergyType : UINT
GET
isEnergyType := m_isEnergyType;
END_GET
END_PROPERTY

PROPERTY kinematicParameters :REFERENCE TO ST_InstruKinematicParam
GET
kinematicParameters ref=m_kinematicParameters;
END_GET
END_PROPERTY

PROPERTY nextScopePosture : E_EndoscopePosture
GET
nextScopePosture:= m_nextEndoscopePosture;
END_GET
SET
m_nextEndoscopePosture := nextScopePosture;
END_SET
END_PROPERTY

PROPERTY nextScopeType : E_EndoscopePosture
GET
nextScopeType:= m_nextEndoscopeType;
END_GET
SET
m_nextEndoscopeType := nextScopeType;
END_SET
END_PROPERTY

PROPERTY onChipData : REFERENCE TO ST_InstruOnChipData
GET
onChipData ref=m_onChipData;
END_GET
END_PROPERTY

METHOD PROTECTED proGrsapForcepsGripAngleFK : BOOL
VAR_INPUT
	frontAngle:LREAL;
END_VAR
VAR_OUTPUT
	endAngle:LREAL;
	Succeed:BOOL;
END_VAR
VAR
	minFrontAng :LREAL  := 16.6*2*g_deg2Rad;
	maxFrontAng :LREAL := 49.18*2*g_deg2Rad;
	AB :LREAL := 2.8;
	BC:LREAL := 5.26;
	Angle_Initial_A:LREAL := 16.6 * g_deg2Rad; 
	SIN_C,Angle_Initial_C,End_Angle_Single,Angle_Inc_C,Angle_C,SIN_A,Angle_A,Angle_Inc_A:LREAL;
END_VAR

//**************已知：器械前端开合角，求解：末端开合角***************//

//输入合法性判断，物理极限是[16.6*2，49.18*2]度
frontAngle := LIMIT(minFrontAng, frontAngle, maxFrontAng);


SIN_C:=AB*SIN(Angle_Initial_A)/BC;
Angle_Initial_C:=ASIN(SIN_C);

Angle_Inc_A:=frontAngle/2;
Angle_A:=Angle_Initial_A+Angle_Inc_A;

SIN_C:=AB*SIN(Angle_A)/BC;
Angle_C:=ASIN(SIN_C);

Angle_Inc_C:=Angle_C-Angle_Initial_C;
endAngle:=Angle_Inc_C*2;
END_METHOD

METHOD PROTECTED proGrsapForcepsGripAngleIK : BOOL
VAR_INPUT
	endAngle:LREAL;
END_VAR
VAR_OUTPUT
	frontAngle:LREAL;
	Succeed:BOOL;
END_VAR
VAR
	minEndAng :LREAL  := 0;
	maxEndAng :LREAL := 38*g_deg2Rad;
	AB :LREAL := 2.8;
	BC:LREAL := 5.26;
	Angle_Initial_A:LREAL := 16.6 * g_deg2Rad; 
	
	SIN_C,Angle_Initial_C,End_Angle_Single,Angle_Inc_C,Angle_C,SIN_A,Angle_A,Angle_Inc_A:LREAL;
END_VAR

//***************已知：器械末端开合角，求解：前端开合角********************//

//输入合法性判断，物理极限是[0,30]度
endAngle:= LIMIT(minEndAng, endAngle, maxEndAng);

SIN_C:=AB*SIN(Angle_Initial_A)/BC;
Angle_Initial_C:=ASIN(SIN_C);

End_Angle_Single:=endAngle/2;
Angle_Inc_C:=End_Angle_Single;
Angle_C:=Angle_Initial_C+Angle_Inc_C;

SIN_A:=BC*SIN(Angle_C)/AB;
Angle_A:=ASIN(SIN_A);

Angle_Inc_A:=Angle_A-Angle_Initial_A;
frontAngle:=Angle_Inc_A*2;
END_METHOD

METHOD PUBLIC readParameters : BOOL
VAR_INPUT
	startFlag :BOOL;
END_VAR

VAR
	paramIdx :INT;
END_VAR
// TODO: read m_kinematic parameters from chip 
//Take the rising edge of the read signal
m_ReadDelay(IN:= m_Step=10, PT:= m_DealyTime, Q=> , ET=> );//计时器
IF startFlag AND m_curReadTries < m_maxReadTries THEN
	m_Step:=0;
	m_onChipData.m_InstruReadSucceed:=FALSE;
	m_onChipData.m_Error:=FALSE;
	m_onChipData.m_ErrorID:=0;
	m_resetArmLEDFlag :=TRUE;
END_IF


CASE m_Step OF
	
	0://向6093发送0x8000  0000---发送读取信号
		m_Value:=16#80000000; 
		m_SdoWrite(sNetId:= m_ArmNetId, nSlaveAddr:= m_JointInstruAddr, nSubIndex:= 0, nIndex:= 16#6093, pSrcBuf:= ADR(m_Value), cbBufLen:= SIZEOF(m_Value), bExecute:= TRUE, );
		IF NOT m_SdoWrite.bBusy THEN
			m_SdoWrite(bExecute:=FALSE);
			m_Step:=10;
		END_IF
		
		
	10://延时0.5s、防止值还没有返回
		IF m_ReadDelay.Q THEN
			m_Step:=20;
		END_IF

		
	20://从6093地址中拿值
		m_SdoRead(sNetId:= m_ArmNetId, nSlaveAddr:= m_JointInstruAddr,	nSubIndex:= 0, nIndex:= 16#6093, pDstBuf:= ADR(m_IDReadResult), cbBufLen:= SIZEOF(m_IDReadResult), bExecute:= TRUE, 	tTimeout:= , bBusy=> , bError=> , nErrId=> , cbRead=> );
		IF NOT m_SdoRead.bBusy THEN
			m_SdoRead(bExecute:=FALSE);
			m_Step:=30;
		END_IF	
		
	
	30://处理器械ID、低16位
		m_IDResult:=UDINT_TO_ULINT(16#0000FFFF AND m_IDReadResult);
		m_Step:=40;
		
		
	40://读取6095、器械序列号
		m_SdoRead(sNetId:= m_ArmNetId, nSlaveAddr:= m_JointInstruAddr,	nSubIndex:= 0, nIndex:= 16#6095, pDstBuf:= ADR(m_SeriesReadResult), cbBufLen:= SIZEOF(m_SeriesReadResult), bExecute:= TRUE, 	tTimeout:= , bBusy=> , bError=> , nErrId=> , cbRead=> );
		IF NOT m_SdoRead.bBusy THEN
			m_SdoRead(bExecute:=FALSE);
			m_Step:=50;
		END_IF	
	
		
	50://处理序列号，低30位
		m_onChipData.m_InstruseriesNum:=SHL(m_IDResult,31)+(16#7FFFFFFF AND m_SeriesReadResult);
		m_onChipData.m_InstruID:=LREAL_TO_INT(FLOOR(lr_in:= m_onChipData.m_InstruseriesNum/EXPT(10,9))); //取十进制前三位为器械ID
		m_Step:=60;
		
		
	60://读取6096---器械零点位置
		m_SdoRead(sNetId:= m_ArmNetId, nSlaveAddr:= m_JointInstruAddr,	nSubIndex:= 0, nIndex:= 16#6096, pDstBuf:= ADR(m_PosReadResult), cbBufLen:= SIZEOF(m_PosReadResult), bExecute:= TRUE, 	tTimeout:= , bBusy=> , bError=> , nErrId=> , cbRead=> );
		IF NOT m_SdoRead.bBusy THEN
			m_SdoRead(bExecute:=FALSE);
			m_Step:=70;
		END_IF	
		
		
	70: //处理位置，L1:0-9位，L2:10-19位，L3:20-29位
		zeroPosDecode(m_PosReadResult, o_q1=>m_onChipData.m_InstruPos[1],o_q2=>m_onChipData.m_InstruPos[2],o_q3=>m_onChipData.m_InstruPos[3]);
		m_onChipData.m_InstruPos[4] := m_jnt4ZeroPos;
		m_onChipData.m_InstruPos[5] := 0;
		
		m_Step:=80;
		
	80://读取器械使用次数 6094
		m_SdoRead(sNetId:= m_ArmNetId, nSlaveAddr:= m_JointInstruAddr,	nSubIndex:= 0, nIndex:= 16#6094, pDstBuf:= ADR(m_UsageReadResult), cbBufLen:= SIZEOF(m_UsageReadResult), bExecute:= TRUE, 	tTimeout:= , bBusy=> , bError=> , nErrId=> , cbRead=> );
		IF NOT m_SdoRead.bBusy THEN
			m_SdoRead(bExecute:=FALSE);
			m_Step:=90;
		END_IF	
		
		
	90://处理器械使用次数读取结果
		m_onChipData.m_InstruusageCounts:=m_UsageReadResult;
		m_InstruUsageToLED:=LIMIT(0,m_UsageReadResult,99);
		m_Step:=100;
		
		
	100://将器械使用次数写入LED
		m_Value:=ULINT_TO_UDINT(16#FFFF AND m_InstruUsageToLED) ;
		m_SdoWrite(sNetId:= m_ArmNetId, nSlaveAddr:= 1003, nSubIndex:= 06, nIndex:= 16#6090, pSrcBuf:= ADR(m_Value), cbBufLen:= SIZEOF(m_Value), bExecute:= TRUE, tTimeout:= , bBusy=> , bError=> , nErrId=> );
		IF NOT m_SdoWrite.bBusy THEN
			m_SdoWrite(bExecute:=FALSE);
			m_Step:=110;
		END_IF
		
	110://处理当器械使用次数达到上限后、在同一场手术中还能使用
		IF m_onChipData.m_InstruusageCounts=m_onChipData.m_InstrumaxUsageCounts THEN		
			//TODO: check this part
			m_InstruSeriesRecord:=InstruIDRecord(i_NewValue:= m_onChipData.m_InstruusageCounts, i_ArrayData:= m_InstruSeriesRecord);
		END_IF
		m_Step:=120;
		
		
	120://结果诊断
		m_onChipData.m_ErrorID:=0;
		m_onChipData.m_InstruReadSucceed:=checkInstruType();
		IF NOT(m_onChipData.m_InstruReadSucceed) THEN
			m_onChipData.m_Error:=TRUE;
			m_onChipData.m_ErrorID:=1;
			
		ELSIF SlaveArmControl.m_slaveRobot.m_endoscopeMounted AND m_instruType = InstruType_Endoscope THEN
			m_onChipData.m_InstruReadSucceed := FALSE;
			m_onChipData.m_Error:=TRUE;
			m_onChipData.m_ErrorID:=3;
			
		ELSIF m_onChipData.m_InstruusageCounts>m_onChipData.m_InstrumaxUsageCounts AND m_onChipData.m_InstruID<>20 THEN
			m_HaveRecord:=InstruSreiesFind(i_NewValue:=m_onChipData.m_InstruseriesNum , i_ArrayData:=m_InstruSeriesRecord );
			IF m_HaveRecord THEN
				//
			ELSE
				m_onChipData.m_InstruReadSucceed := FALSE;
				m_onChipData.m_Error:=TRUE;
				m_onChipData.m_ErrorID:=2;
			END_IF
		END_IF
		m_Step :=-1;
		m_curReadTries := m_curReadTries +1;
	
END_CASE
END_METHOD

METHOD PUBLIC reset : BOOL
VAR_INPUT
END_VAR
VAR
	i:INT;
END_VAR
m_Step := -1;
m_curReadTries := 0;
m_onChipData.m_InstruID := 0;
m_onChipData.m_InstruseriesNum :=0;
m_onChipData.m_Error:=FALSE;
m_onChipData.m_ErrorID:=0;
m_onChipData.m_InstruReadSucceed:=FALSE;
m_isSingleFinger:=FALSE;
m_isEnergyType := 0;
m_instruType:=InstruType_UNKNOWM;
m_instruName := g_instruNullName;
m_instruTypeIdx := 0 ;

FOR i:= 4 TO 8 BY 1 DO
	m_jntPosOffset[i]:=0;
END_FOR

// init joint motion range
FOR i:=1 TO 3 DO
	m_kinematicParameters.m_wristMinDHJntPos[i]:=GVL_SlaveMotorParameters.g_minDHJntPos[i+3];
	m_kinematicParameters.m_wristMaxDHJntPos[i]:=GVL_SlaveMotorParameters.g_maxDHJntPos[i+3];
END_FOR

// reset endoscope type and posture
m_curEndoscopeType :=EndoScopeType_30;
m_nextEndoscopeType :=EndoScopeType_30;
m_curEndoscopePosture :=EndoscopePosture_HeadDown;
m_nextEndoscopePosture :=EndoscopePosture_HeadDown;

//arm LED reset
IF m_resetArmLEDFlag THEN
	m_Value:=0 ;
	m_SdoWrite(sNetId:= m_ArmNetId, nSlaveAddr:= 1003, nSubIndex:= 06, nIndex:= 16#6090, pSrcBuf:= ADR(m_Value), cbBufLen:= SIZEOF(m_Value), bExecute:= TRUE, tTimeout:= , bBusy=> , bError=> , nErrId=> );
END_IF
IF NOT m_SdoWrite.bBusy THEN
	m_SdoWrite(bExecute:=FALSE);
	m_resetArmLEDFlag := FALSE;
END_IF
END_METHOD

PROPERTY resetArmLED : BOOL
SET
m_resetArmLEDFlag := resetArmLED;
END_SET
END_PROPERTY

METHOD ultrasoundKnifeGripAngleFK : LREAL
VAR_INPUT
	// motor joint position of slave arm
	i_jntPos :LREAL;
END_VAR

VAR
	m_jntPos : LREAL;
END_VAR

m_jntPos := i_jntPos;

m_jntPos := LIMIT (-20*g_deg2Rad,m_jntPos,70*g_deg2Rad);

ultrasoundKnifeGripAngleFK := ASIN((m_jntPos*g_uknifeMotorLead * g_uknifeLeverRatio/(2*pi) -  g_uknifeGripTravel * SIN(g_uknifeGripDividAngle))/g_uknifeGripTravel)+g_uknifeGripDividAngle;
END_METHOD

METHOD ultrasoundKnifeGripAngleIK : LREAL
VAR_INPUT
	// gripper angle
	i_gripAngle :LREAL;
END_VAR

VAR
	m_gripAngle : LREAL;
END_VAR

m_gripAngle := i_gripAngle;

ultrasoundKnifeGripAngleIK := (g_uknifeGripTravel * (SIN(g_uknifeGripDividAngle) - SIN(g_uknifeGripDividAngle - m_gripAngle))/(g_uknifeMotorLead*g_uknifeLeverRatio/(2*pi)));
END_METHOD

METHOD writeNumOfUseToChip : BOOL
VAR_INPUT
	startFlag :BOOL;
	i_useNumFromUI :UINT;
END_VAR

writeNumOfUseToChip := FALSE;
m_writeLDP(CLK:= startFlag, Q=> );
m_ReadNumDelay(IN:= m_useNumStep = 10, PT:= m_DealyTime, Q=> , ET=> );
IF m_writeLDP.Q THEN
	m_useNumStep:=0;
END_IF

CASE m_useNumStep OF
	0: 
		m_Value:=16#80000000; 
		m_SdoWrite(sNetId:= m_ArmNetId, nSlaveAddr:= m_JointInstruAddr, nSubIndex:= 0, nIndex:= 16#6094, pSrcBuf:= ADR(m_Value), cbBufLen:= SIZEOF(m_Value), bExecute:= TRUE, );
		IF NOT m_SdoWrite.bBusy THEN
			m_SdoWrite(bExecute:=FALSE);
			m_useNumStep:=10;
		END_IF
	
	10:
		IF m_ReadNumDelay.Q THEN
			m_useNumStep:=20;
		END_IF
		
	20:
		m_SdoRead(sNetId:= m_ArmNetId, nSlaveAddr:= m_JointInstruAddr,	nSubIndex:= 0, nIndex:= 16#6094, pDstBuf:= ADR(m_useNumReadResult), cbBufLen:= SIZEOF(m_useNumReadResult), bExecute:= TRUE, 	tTimeout:= , bBusy=> , bError=> , nErrId=> , cbRead=> );
		IF NOT m_SdoRead.bBusy THEN
			m_SdoRead(bExecute:=FALSE);
			m_useNumStep:=30;
		END_IF
		
	30://Verify the actual usage count and the usage count given by the UI
		IF m_useNumReadResult = i_useNumFromUI THEN
			m_useNumSendToLED := LIMIT(0, m_useNumReadResult, 99);
			m_useNumStep:=40;
		ELSE
			m_useNumStep:=50;
		END_IF
		
	40: 
		m_Value:=ULINT_TO_UDINT( m_useNumSendToLED) ;
		m_SdoWrite(sNetId:= m_ArmNetId, nSlaveAddr:= 1003, nSubIndex:= 06, nIndex:= 16#6090, pSrcBuf:= ADR(m_Value), cbBufLen:= SIZEOF(m_Value), bExecute:= TRUE, tTimeout:= , bBusy=> , bError=> , nErrId=> );
		IF NOT m_SdoWrite.bBusy THEN
			m_SdoWrite(bExecute:=FALSE);
			m_onChipData.m_InstruUsageCounts:=m_useNumReadResult;
			writeNumOfUseToChip := TRUE;
			m_useNumStep:=-1;
		END_IF
		
END_CASE
END_METHOD

METHOD PUBLIC writeZeroPosToChip : BOOL
VAR_INPUT
	i_q1:LREAL;
	i_q2:LREAL;
	i_q3:LREAL;
END_VAR
zeroPosCode(i_q1,i_q2,i_q3, o_code=>m_zeroPosCode);

writeZeroPosToChip:=FALSE;
m_SdoWrite(sNetId:= m_ArmNetId, nSlaveAddr:= m_JointInstruAddr, nSubIndex:= 0, nIndex:= 16#6096, pSrcBuf:= ADR(m_zeroPosCode), cbBufLen:= SIZEOF(m_zeroPosCode), bExecute:= TRUE, );
IF NOT m_SdoWrite.bBusy THEN
	m_SdoWrite(bExecute:=FALSE);
	writeZeroPosToChip:=TRUE;
END_IF
END_METHOD

// code instrument joints(4/5/6) zero position as a UDINT
// joint1 : bit 21-30; joint2: bit 11-20; joint3: bit1-10
// zeroPos: [0, 2pi]; code:[0-3sFF]
METHOD PROTECTED zeroPosCode : BOOL
VAR_INPUT
	i_q1:LREAL;
	i_q2:LREAL;
	i_q3:LREAL;
END_VAR
VAR_OUTPUT
	o_code:UDINT;
END_VAR
VAR
	posCode:UDINT;
END_VAR
// highest bit set to 1
o_code:=2;

// joint1
posCode := LREAL_TO_UDINT(16#3FF * LIMIT(0,i_q1/g_2pi,1));
o_code := SHL(o_code, 10);
o_code := o_code OR posCode;

// joint2
posCode := LREAL_TO_UDINT(16#3FF * LIMIT(0,i_q2/g_2pi,1));
o_code := SHL(o_code, 10);
o_code := o_code OR posCode;

// joint3
posCode := LREAL_TO_UDINT(16#3FF * LIMIT(0,i_q3/g_2pi,1));
o_code := SHL(o_code, 10);
o_code := o_code OR posCode;
END_METHOD

// decode instrument joints(4/5/6) zero position from a UDINT
// joint1 : bit 21-30; joint2: bit 11-20; joint4: bit1-10
// zeroPos: [0, 2pi]; code:[0-2FF]
METHOD PROTECTED zeroPosDecode : BOOL
VAR_INPUT
	i_posCode :UDINT;
END_VAR
VAR_OUTPUT
	o_q1:LREAL;
	o_q2:LREAL;
	o_q3:LREAL;
END_VAR
VAR
	posCode:UDINT;
END_VAR
// joint3
posCode := i_posCode AND 16#3FF;
o_q3 := g_2pi *  posCode/16#3FF;

// joint2
i_posCode := SHR(i_posCode, 10);
posCode := i_posCode AND 16#3FF;
o_q2 := g_2pi *  posCode/16#3FF;

// joint1
i_posCode := SHR(i_posCode, 10);
posCode := i_posCode AND 16#3FF;
o_q1 := g_2pi *  posCode/16#3FF;
END_METHOD

END_FUNCTION_BLOCK

// ---- Mains/SlaveArmControl.TcPOU
PROGRAM SlaveArmControl
VAR
	// master robot data, input from master controller box
	m_masterRobotData AT %I* : MSCommu_MasterStatus;
	
	// all data from other tasks and controller 
	m_slaveInputDataPool : ST_SlaveInputDataPool;
		
	// slave robot data, ouput to master controller box
	m_slaveRobotData AT %Q* :MSCommu_slaveStatus;
	
	// slave robot status, including arm status and cartesian data, output to other tasks
	m_slaveStatus AT%Q* :ST_slaveStatus;
	
	// slave robot joint data, output to other tasks
	m_slaveJointsData AT %Q* :ST_slaveJointData;
	
	// flag to init robot
	m_robotInit :BOOL :=FALSE;
	
	// wait time before robot init  for ethercat to be statble 
	m_robotInitWaitTime : LREAL:=0;
	
	// slave robot
	m_slaveRobot:FB_SlaveRobot;

	// code execute time measure
	m_codeTime : Profiler;
	
END_VAR

m_codeTime(START:=TRUE, RESET:=TRUE);

// wait communication to be stable
IF(m_robotInitWaitTime<g_robotInitWaitTime) THEN
	m_robotInitWaitTime := m_robotInitWaitTime+g_slaveArmCtrlCycleTime;
	RETURN;
END_IF

// robot init
IF m_robotInit =FALSE THEN
	m_slaveRobot.Init();
	m_robotInit:=TRUE;
END_IF

// input from UI
UIInputProcess();

// master input data cast
masterInputDataCast(m_masterRobotData, m_slaveInputDataPool.m_masterStatus);

// robot run
m_slaveRobot.run(m_slaveInputDataPool);

// update data pool
m_slaveRobot.getStatus(m_slaveStatus,m_slaveJointsData);

// slave output data cast
slaveOutputDataCast(m_slaveInputDataPool.m_setupStatus, m_slaveStatus, m_slaveRobotData);

// output to UI
UIOutputProcess();

m_codeTime(START:=FALSE);

// convert from MSCommu_Mastertatus for master-slave communication to local ST_MasterStatus for control
METHOD masterInputDataCast : BOOL
VAR_IN_OUT CONSTANT
	masterInputData:MSCommu_MasterStatus;
END_VAR
VAR_IN_OUT
	masterStatus :ST_MasterStatus;
END_VAR

VAR
	i : INT;
END_VAR
masterStatus.m_masterHeartBeat := masterInputData.m_heartBeat;
masterStatus.m_motionScale := masterInputData.m_motionScale;
masterStatus.m_slaveSelfCheckFlag := masterInputData.m_slaveSelfCheckFlag OR GVL_interactUI.g_salveSelfCheckEnable;
masterStatus.m_masterStopButton := masterInputData.m_masterStopButton;
masterStatus.m_uiResetFault := masterInputData.m_uiResetFault;

FOR i:=1 TO g_mArmNum DO
	masterStatus.m_armState[i] := masterInputData.m_armState[i];
	masterStatus.m_teleSlaveArmIdx[i] :=masterInputData.m_teleSlaveArmIdx[i];
	masterStatus.m_gripAngle[i] := masterInputData.m_gripAngle[i];
	masterStatus.m_curArmPose[i].m_pos := masterInputData.m_curArmPose[i].m_pos;
	masterStatus.m_curArmPose[i].m_rot := masterInputData.m_curArmPose[i].m_rot;
	masterStatus.m_curArmTwist[i] :=masterInputData.m_curArmTwist[i];
	masterStatus.m_pedalHover[i] := masterInputData.m_pedalHover[i];
	masterStatus.m_electricKnifePedalTrigger[i] := masterInputData.m_electricKnifePedalTrigger[i];
	masterStatus.m_tryMSControl[i] := masterInputData.m_tryMSControl[i];
END_FOR
END_METHOD

// convert from local ST_SlaveStatus for control to MSCommu_SlaveStatus for master-slave communication
METHOD slaveOutputDataCast : BOOL
VAR_IN_OUT CONSTANT
	setupStatus :ST_SetupStatus;
	slaveStatus :ST_SlaveStatus;
END_VAR
VAR_IN_OUT 
	slaveOutputData : MSCommu_SlaveStatus;
END_VAR

VAR
	slavePoseInCart, slavePoseInScope:ST_Frame;
	tmpFrame :ST_Frame;
	i :INT;
END_VAR
// Slave heart beat
IF slaveOutputData.m_heartBeat > 10 THEN
	slaveOutputData.m_heartBeat :=0;
ELSE
	slaveOutputData.m_heartBeat :=slaveOutputData.m_heartBeat+1;
END_IF

slaveOutputData.m_seflCheckPass:=  m_slaveInputDataPool.m_UIData.m_armSelfCheckFinshed[1] AND  m_slaveInputDataPool.m_UIData.m_armSelfCheckFinshed[2] AND m_slaveInputDataPool.m_UIData.m_armSelfCheckFinshed[3] AND m_slaveInputDataPool.m_UIData.m_armSelfCheckFinshed[4] ;
slaveOutputData.m_endoscopeMounted :=slaveStatus.m_endoscopeMounted;
slaveOutputData.m_endoscopePose.m_pos :=slaveStatus.m_endoscopePose.m_pos;
slaveOutputData.m_endoscopePose.m_rot :=slaveStatus.m_endoscopePose.m_rot;
slaveOutputData.m_slaveStopButton := NOT SafetyCheck.m_stopButton;

FOR i := 1 TO g_sArmNum DO
	slaveOutputData.m_asepticDeployCompletedFlag := (SlaveArmControl.m_slaveInputDataPool.m_UIData.m_slaveArmDisableFlag[i] OR SlaveArmControl.m_slaveRobot.m_panelMountedFlag[i]) AND m_slaveInputDataPool.m_UIData.m_dumpEnergy >= 30;	
	IF NOT slaveOutputData.m_asepticDeployCompletedFlag THEN
		EXIT;
	END_IF
END_FOR


FOR i:= 1 TO g_sArmNum DO
	slaveOutputData.m_armState[i] := slaveStatus.m_armState[i];
	slaveOutputData.m_instruStauts[i].m_fingerAngle := slaveStatus.m_instruStauts[i].m_fingerAngle;
	slaveOutputData.m_instruStauts[i].m_ready := slaveStatus.m_instruStauts[i].m_ready;
	slaveOutputData.m_instruStauts[i].m_type := slaveStatus.m_instruStauts[i].m_type;
	slaveOutputData.m_instruEnergyType[i] := m_slaveRobot.m_slaveArms[i].m_instrument.isEnergyType;
	slavePoseInCart := transform(setupStatus.m_curEndPose[i], slaveStatus.m_curArmPose[i]);
	tmpFrame :=invFrame(slaveStatus.m_endoscopePose);
	slavePoseInScope := transform(tmpFrame, slavePoseInCart);
	slaveOutputData.m_curArmPose[i].m_pos :=slavePoseInScope.m_pos;
	slaveOutputData.m_curArmPose[i].m_rot :=slavePoseInScope.m_rot;
	slaveOutputData.m_masterSlavePoseError[i] :=slaveStatus.m_masterSlavePoseError[i];
END_FOR
END_METHOD

// tranform data from UI(global variable write by ADS) to ST_UIData
METHOD UIInputProcess : BOOL
VAR_INPUT
END_VAR
VAR
	i:int;
END_VAR
VAR_STAT
	masterSlaveFlag : BOOL:=FALSE;
END_VAR
// arm disable
FOR i:=1 TO g_sArmNum DO 
	m_slaveInputDataPool.m_UIData.m_slaveArmDisableFlag[i]:= FALSE;
END_FOR
IF GVL_interactUI.g_armIsDisable >0 AND GVL_interactUI.g_armIsDisable<= g_sArmNum THEN
	m_slaveInputDataPool.m_UIData.m_slaveArmDisableFlag[GVL_interactUI.g_armIsDisable]:= TRUE;
END_IF
FOR i:=1 TO g_sArmNum DO 
	IF m_slaveRobot.m_slaveArmState[i] = SlaveArmState_MasterSlave THEN
		masterSlaveFlag :=TRUE;
	END_IF
	 
END_FOR
IF masterSlaveFlag THEN
	m_slaveInputDataPool.m_UIData.m_dumpEnergy := 100;
ELSE
	m_slaveInputDataPool.m_UIData.m_dumpEnergy := GVL_interactUI.g_dumpEnergyUPS;
END_IF
END_METHOD

METHOD UIOutputProcess : BOOL
VAR_INPUT
END_VAR

VAR
	i , j: INT;
END_VAR

VAR_STAT
	m_instruUsageCountsLast : ARRAY [1..g_sArmNum] OF ULINT;
END_VAR
//endoscope type
IF m_slaveRobot.m_endoScopeType = EndoscopeType_0  THEN
	GVL_interactUI.g_scopeType:= 0;
ELSIF m_slaveRobot.m_endoScopeType = EndoscopeType_30  THEN
	GVL_interactUI.g_scopeType := 30;
END_IF

//arm state machine
GVL_interactUI.g_armStateMachine.m_stateMachineArm1:=m_slaveStatus.m_armState[1];
GVL_interactUI.g_armStateMachine.m_stateMachineArm2:=m_slaveStatus.m_armState[2];
GVL_interactUI.g_armStateMachine.m_stateMachineArm3:=m_slaveStatus.m_armState[3];
GVL_interactUI.g_armStateMachine.m_stateMachineArm4:=m_slaveStatus.m_armState[4];

//arm is adjustment state
FOR i := 1 TO g_sArmNum BY 1 DO
	IF m_slaveStatus.m_armState[i] = SlaveArmState_Adjust OR SetupArmControl.m_setupStatus.m_armState[i] = SetupArmState_ManualAdjust 
							OR SetupArmControl.m_setupStatus.m_armState[i] = SetupArmState_AutoAdjust THEN
		GVL_interactUI.g_armIsAdjustment[i] := 1;
	ELSE
		GVL_interactUI.g_armIsAdjustment[i] := 0;
	END_IF
END_FOR


//arm self check status
FOR i := 1 TO g_sArmNum DO
	m_slaveInputDataPool.m_UIData.m_armInSelfCheck[i] := m_slaveStatus.m_armState[i] = SlaveArmState_SelfCheck AND NOT m_slaveInputDataPool.m_UIData.m_slaveArmDisableFlag[i];
	m_slaveInputDataPool.m_UIData.m_armSelfCheckFinshed[i] := m_slaveStatus.m_selfCheckPass[i] OR m_slaveInputDataPool.m_UIData.m_slaveArmDisableFlag[i];
END_FOR

IF m_slaveInputDataPool.m_UIData.m_armInSelfCheck[1] OR m_slaveInputDataPool.m_UIData.m_armInSelfCheck[2] OR m_slaveInputDataPool.m_UIData.m_armInSelfCheck[3] OR m_slaveInputDataPool.m_UIData.m_armInSelfCheck[4] THEN
	GVL_interactUI.g_slaveSelfCheckStatus := 1;
ELSIF m_slaveInputDataPool.m_UIData.m_armSelfCheckFinshed[1] AND m_slaveInputDataPool.m_UIData.m_armSelfCheckFinshed[2] AND m_slaveInputDataPool.m_UIData.m_armSelfCheckFinshed[3] AND m_slaveInputDataPool.m_UIData.m_armSelfCheckFinshed[4] THEN
	GVL_interactUI.g_slaveSelfCheckStatus := 2;
ELSE
	GVL_interactUI.g_slaveSelfCheckStatus := 0;
END_IF

//instrument information export to UI
FOR i := 1 TO g_sArmNum DO
	GVL_interactUI.g_instruInformatiom[i].m_instruIsConnected:=m_slaveStatus.m_instruStauts[i].m_ready;
	GVL_interactUI.g_instruInformatiom[i].m_instruInMasterSlave := (m_slaveStatus.m_armState[i] = SlaveArmState_MasterSlave OR m_slaveStatus.m_armState[i] = SlaveArmState_EndoScope);
	IF m_slaveStatus.m_instruStauts[i].m_type = InstruType_Endoscope THEN
		GVL_interactUI.g_instruInformatiom[i].m_instruType := 4;
		GVL_interactUI.g_scopeGravityAngle := m_slaveRobot.m_slaveArms[i].curDHJntPos[4];
	ELSE
		GVL_interactUI.g_instruInformatiom[i].m_instruType := m_slaveRobot.m_slaveArms[i].m_instrument.isEnergyType;
	END_IF
	
	GVL_interactUI.g_instruInformatiom[i].m_armId := i;
	GVL_interactUI.g_instruInformatiom[i].m_instruSerialNum :=  m_slaveRobot.m_slaveArms[i].m_instrument.onChipData.m_InstruseriesNum;
	GVL_interactUI.g_instruInformatiom[i].m_instruID := m_slaveRobot.m_slaveArms[i].m_instrument.onChipData.m_InstruID;
	GVL_interactUI.g_instruInformatiom[i].m_nameEn := m_slaveRobot.m_slaveArms[i].m_instrument.instruName;
	GVL_interactUI.g_instruInformatiom[i].m_nameCh := m_slaveRobot.m_slaveArms[i].m_instrument.instruNameCH;
	
	//instrument pedal hover and pedal active
	GVL_interactUI.g_instruInformatiom[i].m_pedalHover:=FALSE;
	GVL_interactUI.g_instruInformatiom[i].m_pedalActive := 0;
	FOR j := 1 TO g_mArmNum BY 1 DO
		 IF  m_slaveInputDataPool.m_masterStatus.m_teleSlaveArmIdx[j] > 0 AND   m_slaveInputDataPool.m_masterStatus.m_teleSlaveArmIdx[j] <= 4  THEN
			IF m_slaveInputDataPool.m_masterStatus.m_pedalHover[j] = TRUE THEN
				GVL_interactUI.g_instruInformatiom[m_slaveInputDataPool.m_masterStatus.m_teleSlaveArmIdx[j]].m_pedalHover:=TRUE;
			ELSE
				GVL_interactUI.g_instruInformatiom[m_slaveInputDataPool.m_masterStatus.m_teleSlaveArmIdx[j]].m_pedalHover:=FALSE;
			END_IF
			
			IF m_slaveRobot.m_slaveArms[m_slaveInputDataPool.m_masterStatus.m_teleSlaveArmIdx[j]].m_instrument.isEnergyType > 0 THEN
				IF m_slaveInputDataPool.m_masterStatus.m_electricKnifePedalTrigger[j] = 1 THEN 
					GVL_interactUI.g_instruInformatiom[m_slaveInputDataPool.m_masterStatus.m_teleSlaveArmIdx[j]].m_pedalActive := 1;
				ELSIF m_slaveInputDataPool.m_masterStatus.m_electricKnifePedalTrigger[j] = 2 THEN 
					GVL_interactUI.g_instruInformatiom[m_slaveInputDataPool.m_masterStatus.m_teleSlaveArmIdx[j]].m_pedalActive := 2;
				END_IF
			END_IF
			
		END_IF
	END_FOR
	
	//instrument number of  use
	IF m_slaveRobot.m_slaveArms[i].m_instrument.onChipData.m_InstruUsageCounts <> m_InstruUsageCountsLast[i] THEN
		GVL_interactUI.g_instruInformatiom[i].m_useLifeplc := ULINT_TO_UINT(m_slaveRobot.m_slaveArms[i].m_instrument.onChipData.m_InstruUsageCounts);
	END_IF
	m_InstruUsageCountsLast[i] :=m_slaveRobot.m_slaveArms[i].m_instrument.onChipData.m_InstruUsageCounts;
	
	//read-write instrument number of use
	m_slaveRobot.m_slaveArms[i].m_instrument.writeNumOfUseToChip(GVL_interactUI.g_instruInformatiom[i].m_useLifeplc + 1 =  GVL_interactUI.g_instruInformatiom[i].m_useLifeUi AND m_slaveRobot.m_slaveArms[i].m_instrument.onChipData.m_InstruReadSucceed, GVL_interactUI.g_instruInformatiom[i].m_useLifeUi);

	//intrument total number of use
	GVL_interactUI.g_instruInformatiom[i].m_instruTotalLife := m_slaveRobot.m_slaveArms[i].m_instrument.m_instruTotalUse;
	//The coordinates of the instrument relative to the endoscope for UI display
END_FOR
END_METHOD

END_PROGRAM

// ---- FBs_Robots/FB_SlaveRobot.TcPOU
FUNCTION_BLOCK FB_SlaveRobot
VAR_INPUT
END_VAR
VAR_OUTPUT
END_VAR
VAR
	// flag if robot self-check passed
	m_selfCheckPass :ARRAY[1..g_sArmNum] OF BOOL :=[4(false)];
	
	// flag if master are connected
	m_masterOnLine :BOOL :=FALSE;
	m_masterOnLineCheck :FB_masterConnectionCheck;
	
	// master-slave motion scale
	m_motionScale :LREAL;
	
	// index(0 to 4) of slave arm which is tele-linked to master arm
	m_teleSlaveArmIdx :ARRAY[1..g_mArmNum] OF E_MatchedSlaveArmIdx;
	
	// flag if endoscope is mounted
	m_endoscopeMounted :BOOL := FALSE;
	
	// endoscope pose in cart coordinate
	m_endoscopePose : ST_Frame;
	
	// endoscope type 
	m_endoscopeType : E_EndoscopeType:= EndoScopeType_30;
	m_lastEndoScopePostureRobot : E_EndoscopePosture:= EndoScopePosture_HeadDown;
	m_lastEndoScopePostureUI : E_EndoscopePosture:= EndoScopePosture_HeadDown;
	
	// slave arms, responsible for arm kinematic and control
	m_slaveArms :ARRAY[1..g_sArmNum] OF FB_SlaveArm;
	
	// arm state
	m_slaveArmState:ARRAY[1..g_sArmNum] OF E_SlaveArmState:=[4(E_SlaveArmState.SlaveArmState_Error)];
	m_lastSlaveArmState:ARRAY[1..g_sArmNum] OF E_SlaveArmState:=[4(E_SlaveArmState.SlaveArmState_Error)];
	m_nextSlaveArmState:ARRAY[1..g_sArmNum] OF E_SlaveArmState:=[4(E_SlaveArmState.SlaveArmState_Error)];
	
	// matched master arm state
	m_matchedMasterArmState :ARRAY[1..g_sArmNum] OF E_MasterArmState:=[4(E_MasterArmState.MasterArmState_Error)];
	
	// flag if panel and instrument mounted
	m_panelMountedFlag :ARRAY[1..g_sArmNum] OF BOOL :=[4(FALSE)];
	m_instrumentMountedFlag :ARRAY[1..g_sArmNum] OF BOOL :=[4(FALSE)];
	
	// flag if enable instrument invasion after it mounted
	m_instruInvasionEnableFlag :ARRAY[1..g_sArmNum] OF BOOL :=[4(FALSE)];
	
	// all arm controller instance 
	m_armCtrlFactory :ARRAY[1..g_sArmNum,1..SlaveArmState_totalNum] OF I_SlaveArmCtrl;
	m_armError :ARRAY[1..g_sArmNum] OF FB_SlaveCtrlError;
	m_armInit :ARRAY[1..g_sArmNum] OF FB_SlaveCtrlInit;
	m_armSelfCheck :ARRAY[1..g_sArmNum] OF FB_SlaveCtrlSelfCheck;
	m_armStandBy :ARRAY[1..g_sArmNum] OF FB_SlaveCtrlStandBy;
	m_mountPanel :ARRAY[1..g_sArmNum] OF FB_SlaveCtrlMountPanel;
	m_panelReady :ARRAY[1..g_sArmNum] OF FB_SlaveCtrlPanelReady;
	m_mountInstru :ARRAY[1..g_sArmNum] OF FB_SlaveCtrlMountInstru;
	m_instruReady :ARRAY[1..g_sArmNum] OF FB_SlaveCtrlInstruReady;
	m_armMasterSlave :ARRAY[1..g_sArmNum] OF FB_SlaveCtrlMasterSlave;
	m_scopeReady :ARRAY[1..g_sArmNum] OF FB_SlaveCtrlScopeReady;
	m_armEndoscope :ARRAY[1..g_sArmNum] OF FB_SlaveCtrlEndoscope;
	m_armAdjust :ARRAY[1..g_sArmNum] OF FB_SlaveCtrlAdjust;
	m_armPackage :ARRAY[1..g_sArmNum] OF FB_SlaveCtrlPackage;
	m_armCart :ARRAY[1..g_sArmNum] OF FB_SlaveCtrlCart;
	m_armGraCali :ARRAY[1..g_sArmNum] OF FB_SlaveCtrlGraCali;
	m_armTest :ARRAY[1..g_sArmNum] OF FB_SlaveCtrlTest;
	m_instruRetract :ARRAY[1..g_sArmNum] OF FB_SlaveCtrlInstruRetract;
	m_instruInvasion :ARRAY[1..g_sArmNum] OF FB_SlaveCtrlInstruInvasion;
	m_armDisable :ARRAY[1..g_sArmNum] OF FB_SlaveCtrlDisable;
	m_instruCali :ARRAY[1..g_sArmNum] OF FB_SlaveCtrlInstruCali;
	m_scopeToggle :ARRAY[1..g_sArmNum] OF FB_SlaveCtrlScopeToggle;
	m_Performance :ARRAY[1..g_sArmNum] OF FB_SlaveCtrlPerformance;
	m_armStop :ARRAY[1..g_sArmNum] OF FB_SlaveCtrlStop;
	
	// arm controller interface
	m_armCtrl :ARRAY[1..g_sArmNum] OF I_SlaveArmCtrl;
	m_armCtrlCmds :ARRAY[1..g_sArmNum] OF ST_SlaveArmCtrlCmds;

END_VAR

METHOD PROTECTED controllerTransit : BOOL
VAR_INPUT
END_VAR
VAR
	i:int;
END_VAR
FOR i:=1 TO g_sArmNum DO 
	// Controller transit
	IF m_nextSlaveArmState[i]<> m_slaveArmState[i] THEN
		// reset current controller
		m_armCtrl[i].reset();
		
		// transit to new controller
		m_lastSlaveArmState[i]:=m_slaveArmState[i];
		m_slaveArmState[i]:=m_nextSlaveArmState[i];
		m_armCtrl[i]:=m_armCtrlFactory[i,m_slaveArmState[i]];
		
		// init next controller
		m_armCtrl[i].Init(m_slaveArms[i],m_armCtrlCmds[i]);
		m_slaveArms[i].updateCmds(m_armCtrlCmds[i]);
	END_IF
END_FOR
END_METHOD

METHOD PUBLIC getStatus : BOOL
VAR_IN_OUT
	// slave robot information, including arm status and cartesian data
	r_slaveStatus :ST_SlaveStatus;
	
	// slave robot joint data
	r_slaveJointsData :ST_SlaveJointData;
	
END_VAR

VAR
	i:INT;
END_VAR
r_slaveStatus.m_armState:=m_slaveArmState;
r_slaveStatus.m_endoscopeMounted :=m_endoscopeMounted;
r_slaveStatus.m_endoscopePose :=m_endoscopePose;

FOR i:=1 TO g_sArmNum DO
	r_slaveStatus.m_selfCheckPass[i] := m_selfCheckPass[i];	

	// instrument data
	r_slaveStatus.m_instruStauts[i].m_type:=m_slaveArms[i].instrument.m_instruType;
	r_slaveStatus.m_instruStauts[i].m_ready:=m_instrumentMountedFlag[i];
	r_slaveStatus.m_instruStauts[i].m_fingerAngle:=m_slaveArms[i].curGripAngle;
	r_slaveStatus.m_instruReadErrId[i] := m_slaveArms[i].instrument.onChipData.m_ErrorID;
	r_slaveStatus.m_instruInstallStatus[i] := m_slaveArms[i].instruOn;
	r_slaveStatus.m_instruClampErrId[i] := m_mountInstru[i].instruClampErrId;
	r_slaveStatus.m_panelInstallStatus[i] := m_slaveArms[i].panelOn;
	r_slaveStatus.m_panelClampErrId[i] := m_mountPanel[i].panelClampErrId;
	r_slaveStatus.m_trocarOnFlag[i] := m_slaveArms[i].trocarOn;
	r_slaveStatus.m_masterOnLine := m_masterOnLine;
	// cartesion
	r_slaveStatus.m_curArmPose[i]:=m_slaveArms[i].curCartPose;
	r_slaveStatus.m_simArmPose[i]:=m_slaveArms[i].simCartPose;
	r_slaveStatus.m_masterSlavePoseError[i] := m_armMasterSlave[i].masterSlavePoseErr;
	// joint
	r_slaveJointsData.m_curMotorPos[i]:=m_slaveArms[i].curMotorPos;
	r_slaveJointsData.m_curLinkPos[i]:=m_slaveArms[i].curLinkPos;
	r_slaveJointsData.m_curJntPos[i]:=m_slaveArms[i].curJntPos;
	r_slaveJointsData.m_curJntVel[i]:=m_slaveArms[i].curJntVel;
	r_slaveJointsData.m_rawJntCurrent[i] := m_slaveArms[i].rawJntCurrent;
	// command info
	// cartesion
	r_slaveStatus.m_cmdArmPose[i]:=m_slaveArms[i].cmdCartPose;
	// joint info
	r_slaveJointsData.m_cmdJntPos[i]:=m_slaveArms[i].cmdJntPos;
	
END_FOR
END_METHOD

METHOD PUBLIC Init : BOOL
VAR_INPUT
END_VAR
VAR
	i:INT;
END_VAR
FOR i:=1 TO g_sArmNum DO
	// arm init
	m_slaveArms[i].Init(i);
	m_slaveArmState[i]:=SlaveArmState_Init;
	m_lastSlaveArmState[i]:=SlaveArmState_Init;
	m_nextSlaveArmState[i]:=SlaveArmState_Init;
	m_selfCheckPass[i]:=false;
	
	// command init
	m_armCtrlCmds[i].m_jntEnableFlag := g_zeroVec8i;
	m_armCtrlCmds[i].m_jntOPMode := g_slaveAllPosMode;
	m_armCtrlCmds[i].m_cmdCartPose := m_slaveArms[i].curCartPose;
	m_armCtrlCmds[i].m_cmdCartTwist := g_zeroVec6d;
	m_armCtrlCmds[i].m_cmdJntPos := m_slaveArms[i].curJntPos;
	m_armCtrlCmds[i].m_cmdJntVel := g_zeroVec8d;
	m_armCtrlCmds[i].m_cmdJntAcc := g_zeroVec8d;
	m_armCtrlCmds[i].m_cmdJntTrq := g_zeroVec8d;
	
	// generate controller factory
	m_armCtrlFactory[i,SlaveArmState_Error] := m_armError[i];
	m_armCtrlFactory[i,SlaveArmState_Init] := m_armInit[i];
	m_armCtrlFactory[i,SlaveArmState_SelfCheck] := m_armSelfCheck[i];
	m_armCtrlFactory[i,SlaveArmState_Standby] := m_armStandBy[i];
	m_armCtrlFactory[i,SlaveArmState_MountPanel] := m_mountPanel[i];
	m_armCtrlFactory[i,SlaveArmState_PanelReady] := m_panelReady[i];
	m_armCtrlFactory[i,SlaveArmState_MountInstru] := m_mountInstru[i];
	m_armCtrlFactory[i,SlaveArmState_InstruReady] := m_instruReady[i];
	m_armCtrlFactory[i,SlaveArmState_MasterSlave] := m_armMasterSlave[i];
	m_armCtrlFactory[i,SlaveArmState_ScopeReady] := m_scopeReady[i];
	m_armCtrlFactory[i,SlaveArmState_EndoScope] := m_armEndoscope[i];
	m_armCtrlFactory[i,SlaveArmState_Adjust] := m_armAdjust[i];
	m_armCtrlFactory[i,SlaveArmState_Package] := m_armPackage[i];
	m_armCtrlFactory[i,SlaveArmState_Cart] := m_armCart[i];
	m_armCtrlFactory[i,SlaveArmState_GravityCali] := m_armGraCali[i];
	m_armCtrlFactory[i,SlaveArmState_Test] := m_armTest[i];
	m_armCtrlFactory[i,SlaveArmState_InstruRetract] := m_instruRetract[i];
	m_armCtrlFactory[i,SlaveArmState_InstruInvasion] := m_instruInvasion[i];
	m_armCtrlFactory[i,SlaveArmState_Disable] := m_armDisable[i];
	m_armCtrlFactory[i,SlaveArmState_InstruCali] := m_instruCali[i];
	m_armCtrlFactory[i,SlaveArmState_ScopeToggle] := m_scopeToggle[i];
	m_armCtrlFactory[i,SlaveArmState_Performance] := m_Performance[i];
	m_armCtrlFactory[i,SlaveArmState_Stop] := m_armStop[i];
	
	// assign controller
	m_armCtrl[i]:=m_armCtrlFactory[i,m_slaveArmState[i]];
	m_armCtrl[i].Init(m_slaveArms[i],m_armCtrlCmds[i]);
END_FOR
END_METHOD

METHOD PUBLIC run : BOOL
VAR_IN_OUT CONSTANT
	i_slaveInputDataPool:ST_SlaveInputDataPool;
END_VAR
VAR
	i:INT;
END_VAR
m_motionScale := i_slaveInputDataPool.m_masterStatus.m_motionScale;
m_teleSlaveArmIdx := i_slaveInputDataPool.m_masterStatus.m_teleSlaveArmIdx;

// check master connection
m_masterOnLine := m_masterOnLineCheck.check(i_slaveInputDataPool.m_masterStatus.m_masterHeartBeat);

// check if endoscope is mounted
m_endoscopeMounted := FALSE;
FOR i:=1 TO g_sArmNum DO 
	IF m_slaveArms[i].instrument.m_instruType=InstruType_endoscope THEN
		m_endoscopeMounted := TRUE;
		m_endoscopePose := transform(i_slaveInputDataPool.m_setupStatus.m_curEndPose[i], m_slaveArms[i].curCartPose);
		m_endoScopeType := m_slaveArms[i].instrument.curScopeType;
		
		//set endoscope  posture from UI data
		updateScopeUIInfo();
	END_IF
END_FOR

// update arm status
FOR i:=1 TO g_sArmNum DO
	// update dynamic data
	m_slaveArms[i].updateDyna(i_slaveInputDataPool.m_slaveDynaData);
								
	// update slave arm kinematics
	m_slaveArms[i].updateStatus();
END_FOR

// state machine transition
stateMachine(i_slaveInputDataPool);

// controller transition
controllerTransit();

// run arm controller
FOR i:=1 TO g_sArmNum DO
	// null ptr check
	ASSERT(0 <> m_armCtrl[i]);
	
	// run controller
	m_armCtrl[i].run(m_endoscopePose, i_slaveInputDataPool.m_MasterStatus,
					i_slaveInputDataPool.m_setupStatus, m_SlaveArms[i],m_armCtrlCmds[i]);

	// update commands to drivers
	m_slaveArms[i].updateCmds(m_armCtrlCmds[i]);
END_FOR
END_METHOD

// state machine check and transit 
METHOD PROTECTED stateMachine : BOOL
VAR_IN_OUT CONSTANT
		i_slavesInputDataPool:ST_SlaveInputDataPool;
END_VAR
VAR
	i,j:INT;
END_VAR
// check instrument state
FOR i:=1 TO g_sArmNum DO
	// statues check
	IF m_slaveArms[i].panelOn = FALSE THEN
		m_panelMountedFlag[i]:=FALSE;
	END_IF
	IF m_slaveArms[i].instruOn = FALSE THEN
		m_instrumentMountedFlag[i]:=FALSE;			
	END_IF
END_FOR

// get matched master arm state
FOR i:=1 TO g_sArmNum DO 
	m_matchedMasterArmState[i]:=MasterArmState_Error;
	FOR j:=1 TO g_mArmNum DO 
		IF i = i_slavesInputDataPool.m_masterStatus.m_teleSlaveArmIdx[j] THEN
			m_matchedMasterArmState[i] := i_slavesInputDataPool.m_masterStatus.m_armState[j];
		END_IF
	END_FOR
END_FOR

// check if to enable instrument invasion 
FOR i:=1 TO g_sArmNum DO
	IF SlaveArmState_Adjust = m_slaveArmState[i] OR SlaveArmState_Cart = m_slaveArmState[i] OR i_slavesInputDataPool.m_setupStatus.m_armState[i] = SetupArmState_ManualAdjust OR
	    m_slaveArms[i].instrument.instruType = InstruType_Endoscope	 THEN
		m_instruInvasionEnableFlag[i]:=FALSE;
		m_slaveArms[i].resetInstruDepth();
	ELSIF m_instrumentMountedFlag[i] AND m_slaveArms[i].instrument.instruType <> InstruType_Endoscope AND m_slaveArmState[i] <> SlaveArmState_InstruInvasion THEN
		m_instruInvasionEnableFlag[i]:=TRUE;
		m_slaveArms[i].setInstruDepth();
	END_IF
END_FOR  

// state machine transit
FOR i:=1 TO g_sArmNum DO
	CASE m_slaveArmState[i] OF
		// error
		SlaveArmState_Error:
			IF FALSE = i_slavesInputDataPool.m_safetyData.m_slaveErrFlag[i] THEN
				// to standby
				IF m_selfCheckPass[i] THEN
					m_nextSlaveArmState[i] :=SlaveArmState_Standby;
				// to init
				ELSE
					m_nextSlaveArmState[i] :=SlaveArmState_Init;
				END_IF
			END_IF
			// to adjust
			IF (m_slaveArms[i].adjustOn) THEN
				m_nextSlaveArmState[i]:=SlaveArmState_Adjust;
			END_IF
			
		// init
		SlaveArmState_Init:
			m_selfCheckPass[i]:=FALSE;
			m_slaveArms[i].instrument.resetArmLED :=TRUE;
			// to selfcheck
			IF m_armCtrl[i].isFinished AND i_slavesInputDataPool.m_masterStatus.m_slaveSelfCheckFlag  THEN
				m_nextSlaveArmState[i]:=SlaveArmState_SelfCheck;
			// to adjust
			ELSIF m_slaveArms[i].adjustOn THEN
				m_nextSlaveArmState[i]:=SlaveArmState_Adjust;
			END_IF

		//self check
		SlaveArmState_SelfCheck:
			// to standby
			IF m_armCtrl[i].isFinished  THEN
				m_nextSlaveArmState[i]:=SlaveArmState_Standby;
				m_selfCheckPass[i]:=TRUE;
			END_IF
		
		//standby
		SlaveArmState_Standby:
			// to mount panel
			IF m_slaveArms[i].panelOn THEN 
				IF m_panelMountedFlag[i] THEN
					m_nextSlaveArmState[i]:=SlaveArmState_PanelReady;
				ELSE
					m_nextSlaveArmState[i]:=SlaveArmState_MountPanel;
				END_IF
			// to adjust
			ELSIF m_slaveArms[i].adjustOn THEN
				m_nextSlaveArmState[i]:=SlaveArmState_Adjust;
			END_IF
		
		//mount panel
		SlaveArmState_MountPanel:
			// to panel ready
			IF m_armCtrl[i]. isFinished THEN
				m_nextSlaveArmState[i]:=SlaveArmState_PanelReady;
				m_panelMountedFlag[i] :=TRUE;
				
			// to standby
			ELSIF NOT(m_slaveArms[i].panelOn) THEN
				m_nextSlaveArmState[i]:=SlaveArmState_Standby;
			END_IF
		
		//panel ready
		SlaveArmState_PanelReady:
			// to adjust
			IF (m_slaveArms[i].adjustOn) THEN
				m_nextSlaveArmState[i]:=SlaveArmState_Adjust;
			// to stand by
			ELSIF NOT(m_slaveArms[i].panelOn) THEN
				m_nextSlaveArmState[i]:=SlaveArmState_Standby;
			ELSIF m_slaveArms[i].instruOn   THEN
				IF m_instrumentMountedFlag[i] THEN
					// to scope ready
					IF  InstruType_endoscope = m_slaveArms[i].instrument.m_instruType AND m_slaveArms[i].instruReady() THEN 
						m_nextSlaveArmState[i]:=SlaveArmState_ScopeReady;
					// to scope toggle
					ELSIF  InstruType_endoscope = m_slaveArms[i].instrument.m_instruType AND 
								(m_slaveArms[i].instrument.curScopePosture <> m_slaveArms[i].instrument.nextScopePosture OR
								m_slaveArms[i].instrument.curScopeType <> m_slaveArms[i].instrument.nextScopeType) THEN
						m_nextSlaveArmState[i] := SlaveArmState_ScopeToggle;
					// to instrument ready
					ELSIF  m_slaveArms[i].instruReady() THEN
						m_nextSlaveArmState[i]:=SlaveArmState_InstruReady;
					END_IF
				// to mount instrument/endoscope
				ELSIF m_slaveArms[i].readyForInstruMount() THEN
					m_nextSlaveArmState[i]:=SlaveArmState_MountInstru;
				END_IF
			// to instrument retract
			ELSIF  NOT(m_slaveArms[i].readyForInstruMount())  THEN
				m_nextSlaveArmState[i]:=SlaveArmState_InstruRetract;
			END_IF
			
		//mount instrument
		SlaveArmState_MountInstru:
			// to panel ready
			IF NOT(m_slaveArms[i].instruOn)  THEN
				m_nextSlaveArmState[i]:=SlaveArmState_PanelReady;
			ELSIF m_armCtrl[i].isFinished THEN
				m_instrumentMountedFlag[i] :=TRUE;
				
				// to instrument invasion
				IF m_instruInvasionEnableFlag[i] THEN
					m_nextSlaveArmState[i] := SlaveArmState_InstruInvasion;
				// to panel ready
				ELSE
					m_nextSlaveArmState[i]:=SlaveArmState_PanelReady;
				END_IF
				
			END_IF
		
		// instrument ready
		SlaveArmState_InstruReady:
			// to instrument retract
			IF  NOT(m_slaveArms[i].instruOn)  THEN
				m_nextSlaveArmState[i]:=SlaveArmState_InstruRetract;
			// to Adjust
			ELSIF (m_slaveArms[i].adjustOn) THEN
				m_nextSlaveArmState[i]:=SlaveArmState_Adjust;
			// to master-slave
			ELSIF MasterArmState_MasterSlave = m_matchedMasterArmState[i] THEN
				m_nextSlaveArmState[i] := SlaveArmState_MasterSlave;
			END_IF
		
		//master slave control
		SlaveArmState_MasterSlave:
			// to Adjust
			IF (m_slaveArms[i].adjustOn) THEN
				m_nextSlaveArmState[i]:=SlaveArmState_Adjust;
			// to stop
			ELSIF MasterArmState_MasterSlave <> m_matchedMasterArmState[i] OR m_armCtrl[i].isFinished THEN
				m_nextSlaveArmState[i]:=SlaveArmState_Stop;
				m_armStop[i].setInstruBacklash(m_armMasterSlave[i].InstruBacklash);
			// to instrument retract
			ELSIF  NOT(m_slaveArms[i].panelOn) OR NOT(m_slaveArms[i].instruOn) THEN
				m_nextSlaveArmState[i]:=SlaveArmState_InstruRetract;
			END_IF
		
		//endoscope ready
		SlaveArmState_ScopeReady:
			// to instrument retract
			IF NOT(m_slaveArms[i].instruOn) THEN
				m_nextSlaveArmState[i]:=SlaveArmState_InstruRetract;
			// to Adjust
			ELSIF (m_slaveArms[i].adjustOn) THEN
				m_nextSlaveArmState[i]:=SlaveArmState_Adjust;
			// to scope toggle
			ELSIF m_slaveArms[i].instrument.curScopePosture <> m_slaveArms[i].instrument.nextScopePosture OR
					m_slaveArms[i].instrument.curScopeType <> m_slaveArms[i].instrument.nextScopeType THEN
				m_nextSlaveArmState[i] := SlaveArmState_ScopeToggle;
			// to endoscope control
			ELSIF MasterArmState_Endoscope = i_slavesInputDataPool.m_masterStatus.m_armState[1] AND 
				  MasterArmState_Endoscope = i_slavesInputDataPool.m_masterStatus.m_armState[2] THEN
				m_nextSlaveArmState[i] := SlaveArmState_EndoScope;
			END_IF
		
		//endoscope control
		SlaveArmState_EndoScope:
			// to Adjust
			IF (m_slaveArms[i].adjustOn) THEN
				m_nextSlaveArmState[i]:=SlaveArmState_Adjust;
			// to stop
			ELSIF MasterArmState_Endoscope <> i_slavesInputDataPool.m_masterStatus.m_armState[1]
				OR MasterArmState_Endoscope <> i_slavesInputDataPool.m_masterStatus.m_armState[2] THEN
				m_nextSlaveArmState[i]:=SlaveArmState_Stop;
			// to scope toggle
			ELSIF m_slaveArms[i].instrument.curScopePosture <> m_slaveArms[i].instrument.nextScopePosture OR
					m_slaveArms[i].instrument.curScopeType <> m_slaveArms[i].instrument.nextScopeType THEN
				m_nextSlaveArmState[i] := SlaveArmState_ScopeToggle;
			// to instrument retract
			ELSIF  NOT(m_slaveArms[i].panelOn) OR NOT(m_slaveArms[i].instruOn) THEN
				m_nextSlaveArmState[i]:=SlaveArmState_InstruRetract;
			END_IF
			
		//arm adjust
		SlaveArmState_Adjust:
			IF m_slaveArms[i].adjustFallEdge AND m_armCtrl[i].timePeriod > 0.25 THEN
				// to init
				IF NOT (m_selfCheckPass[i]) THEN
					m_nextSlaveArmState[i] :=SlaveArmState_Init;
				// to standby
				ELSE
					m_nextSlaveArmState[i] :=SlaveArmState_Standby;
				END_IF
			END_IF
		
		//scope toggle
		SlaveArmState_ScopeToggle:
			// to instrument retract
			IF NOT(m_slaveArms[i].instruOn) THEN
				m_nextSlaveArmState[i]:=SlaveArmState_InstruRetract;
			// to standby
			ELSIF m_armCtrl[i].isFinished THEN
				m_nextSlaveArmState[i] :=SlaveArmState_Standby;
			END_IF
		
		// package
		SlaveArmState_Package:
			// to Adjust
			IF (m_slaveArms[i].adjustOn) THEN
				m_nextSlaveArmState[i]:=SlaveArmState_Adjust;
			// to standby
			ELSIF m_armCtrl[i].isFinished THEN
				m_nextSlaveArmState[i]:=SlaveArmState_Standby;
			END_IF
			
		// Cart
		SlaveArmState_Cart:
		
		// Gravity Calibration
		SlaveArmState_GravityCali:
			// to Adjust
			IF (m_slaveArms[i].adjustOn) THEN
				m_nextSlaveArmState[i]:=SlaveArmState_Adjust;
			// to standby
			ELSIF m_armCtrl[i].isFinished THEN
				m_nextSlaveArmState[i]:=SlaveArmState_Standby;
			END_IF
			
		//arm test
		SlaveArmState_Test:
			// to stop
			IF  m_armCtrl[i].isFinished THEN
				m_nextSlaveArmState[i]:=SlaveArmState_Stop;
			END_IF
		
		//arm Performance
		SlaveArmState_Performance:
			// to standby
			IF  m_armCtrl[i].isFinished THEN
				m_nextSlaveArmState[i]:=SlaveArmState_Standby;
			END_IF		
			
		//arm stop
		SlaveArmState_Stop:
			// to standby
			IF  m_armCtrl[i].isFinished THEN
				m_nextSlaveArmState[i]:=SlaveArmState_Standby;
			END_IF
		
		// instrument retract
		SlaveArmState_InstruRetract:
			// to Adjust
			IF (m_slaveArms[i].adjustOn) THEN
				m_nextSlaveArmState[i]:=SlaveArmState_Adjust;
			// to standby
			ELSIF m_armCtrl[i].isFinished THEN
				m_nextSlaveArmState[i]:=SlaveArmState_Standby;
			END_IF
		
		// instrument invasion
		SlaveArmState_InstruInvasion:
			// to instrument retract
			IF NOT m_slaveArms[i].instruOn THEN
				m_nextSlaveArmState[i]:=SlaveArmState_InstruRetract;
			// to Adjust
			elsIF (m_slaveArms[i].adjustOn) THEN
				m_nextSlaveArmState[i]:=SlaveArmState_Adjust;
			// to instrument ready
			ELSIF m_armCtrl[i].isFinished THEN
			// to panel ready
				m_nextSlaveArmState[i]:=SlaveArmState_PanelReady;
			END_IF
		
		// arm disable
		SlaveArmState_Disable:
			IF NOT(i_slavesInputDataPool.m_UIData.m_slaveArmDisableFlag[i]) THEN
				// to standby
				IF m_selfCheckPass[i] THEN
					m_nextSlaveArmState[i] :=SlaveArmState_Standby;
				// to init
				ELSE
					m_nextSlaveArmState[i] :=SlaveArmState_Init;
				END_IF
			END_IF
	END_CASE
	
	// control is forbidden if setup arm is not in Hold
	IF SetupArmState_Hold <> i_slavesInputDataPool.m_setupStatus.m_armState[i] AND
		(SlaveArmState_InstruReady = m_nextSlaveArmState[i] OR SlaveArmState_MasterSlave = m_nextSlaveArmState[i]
		 OR SlaveArmState_ScopeReady = m_nextSlaveArmState[i] OR SlaveArmState_EndoScope = m_nextSlaveArmState[i]) THEN
		m_nextSlaveArmState[i]:=SlaveArmState_Standby;
	END_IF
	
	// arm disable
	IF i_slavesInputDataPool.m_UIData.m_slaveArmDisableFlag[i] THEN
		m_nextSlaveArmState[i] := SlaveArmState_Disable;
	// error check
	ELSIF i_slavesInputDataPool.m_safetyData.m_slaveErrFlag[i] AND NOT m_slaveArms[i].adjustOn THEN
		m_nextSlaveArmState[i]:=SlaveArmState_Error;
	END_IF
END_FOR
END_METHOD

METHOD PROTECTED updateScopeUIInfo : BOOL
VAR_INPUT
END_VAR
VAR
	i:INT;
END_VAR
// check if endoscope is mounted
FOR i:=1 TO g_sArmNum DO 
	IF m_slaveArms[i].instrument.m_instruType=InstruType_endoscope THEN
		
		// update command endoscope posture from UI
		IF GVL_interactUI.g_scopeUpDown <> m_lastEndoScopePostureUI AND m_slaveArms[i].instrument.curScopeType = EndoScopeType_30 THEN
			IF GVL_interactUI.g_scopeUpDown = 1 THEN
				m_slaveArms[i].instrument.nextScopePosture := EndoScopePosture_HeadDown;
			ELSIF  GVL_interactUI.g_scopeUpDown = 2 THEN
				m_slaveArms[i].instrument.nextScopePosture := EndoscopePosture_HeadUp;
			END_IF
		END_IF
		
		// update current endoscope posture to UI
		IF m_slaveArms[i].instrument.curScopePosture <> m_lastEndoScopePostureRobot THEN
			IF m_slaveArms[i].instrument.curScopePosture = EndoScopePosture_HeadDown THEN
				GVL_interactUI.g_scopeUpDown := 1 ;
			ELSIF  m_slaveArms[i].instrument.curScopePosture = EndoScopePosture_HeadUp THEN
				GVL_interactUI.g_scopeUpDown := 2;
			END_IF
		END_IF
		m_lastEndoScopePostureRobot := m_slaveArms[i].instrument.curScopePosture;
		
	END_IF
END_FOR

m_lastEndoScopePostureUI := GVL_interactUI.g_scopeUpDown;
END_METHOD

END_FUNCTION_BLOCK

// ---- FBs_SlaveControllers/FB_SlaveCtrlSelfCheck.TcPOU
// Brief: Slave Arm Run Self-check Trajectory
FUNCTION_BLOCK PUBLIC FB_SlaveCtrlSelfCheck EXTENDS FB_SlaveArmCtrlBase
VAR CONSTANT
	m_selfCheckMotionNum :INT :=1;
END_VAR
VAR
	// slave self-check motion parameters
	m_selfCheckPosture:ARRAY [1..m_selfCheckMotionNum, 1..g_sJntNum] OF LREAL:=[0.0, 	-PI/2, GVL_SlaveMotorParameters.g_maxDHJntPos[3], 	5(-g_2pi)];																			//PI/4, -PI/4, 0.3, pi, pi, pi, pi, pi];
	m_selfCheckMaxjntVel:Vec8d:=[0.2, 0.2, 0.1, 5(2.0)];
	m_selfCheckMaxjntAcc:Vec8d:=[1.0, 1.0, 0.5, 5(4.0)];
	m_selfCheckMaxjntJerk:Vec8d:=[2.0,2.0, 1.0, 5(8.0)];
	
	m_selfCheckTrajIdx: INT := 1;
	m_slefCheckPlanner: ARRAY[1..m_selfCheckMotionNum] OF FB_TrajMoveJ;
	
   // wait time for joint enable
   m_enableWaitTime :LREAL := 1.0;

   // time gap between enable and motion
   m_jntMotionTimeGap :LREAL := 0.5;

	
END_VAR

// override this function in each exact controller
METHOD PROTECTED calcCmdJntPos : BOOL
VAR_IN_OUT CONSTANT
	i_endoscopePose : ST_Frame;
	i_masterStatus :ST_MasterStatus;
	i_setupStatus: ST_SetupStatus;
	i_slaveArm :FB_SlaveArm;
END_VAR

VAR 
	i :INT;
	curJntVel :Vec8d;
END_VAR
// check if planner is ready
IF m_slefCheckPlanner[m_selfCheckTrajIdx].isGene = FALSE THEN
	calcCmdJntPos:=FALSE;
	RETURN;
END_IF

// arms enable successively
IF m_timePeriod > m_enableWaitTime THEN
       m_jntEnableFlag :=g_onesVec8i;
END_IF

IF m_timePeriod < m_enableWaitTime + m_jntMotionTimeGap THEN
	RETURN;
END_IF

// traj plan
calcCmdJntPos :=m_slefCheckPlanner[m_selfCheckTrajIdx].evaluate(m_timePeriod-m_enableWaitTime-m_jntMotionTimeGap, jntPos=> m_cmdJntPos, jntVel=>m_cmdJntVel, jntAcc=> m_cmdJntAcc);

// check if to transit to next segment
curJntVel :=i_slaveArm.curJntVel;
IF(m_timePeriod - m_enableWaitTime - m_jntMotionTimeGap > m_slefCheckPlanner[m_selfCheckTrajIdx].duration  AND norm(curJntVel)<7*GVL_SlaveControlParameters.g_jntStaticVelThres) THEN
	m_selfCheckTrajIdx:=m_selfCheckTrajIdx+1;
	m_timePeriod:=0;
END_IF

// check if to terminated
IF(m_selfCheckTrajIdx > m_selfCheckMotionNum) THEN
	m_isFinished:=TRUE;
END_IF
END_METHOD

METHOD PUBLIC init : BOOL
VAR_IN_OUT CONSTANT
	i_slaveArm	:FB_SlaveArm;
END_VAR
VAR_IN_OUT 
	r_slaveArmCtrlCmd :ST_SlaveArmCtrlCmds;
END_VAR

VAR
	i,j :INT;
	startJntPos,endJntPos :Vec8d;
	baseJntPos:Vec8d;
	cycleNum :LREAL;
END_VAR
SUPER^.Init(i_slaveArm,r_slaveArmCtrlCmd);
//m_jntEnableFlag :=g_zeroVec8i;

//set different wait time for each arm, so the arms would run self-check successively
m_enableWaitTime := i_slaveArm.armIdx-1;

// determine base joint position for instrument joint
baseJntPos :=g_zeroVec8d;
FOR i:=4 TO g_sJntNum DO
	cycleNum := FLOOR(i_slaveArm.curJntPos[i]/g_2pi);
	baseJntPos[i]:=cycleNum* g_2Pi;
END_FOR

// traj plan
// fisrt segment
// TODO: joint1/2 stay still in case arms collision
m_selfCheckTrajIdx :=1;
startJntPos:=i_slaveArm.curJntPos;
endJntPos:=startJntPos;
FOR j:=3 TO g_sJntNum DO 
	endJntPos[j]:=baseJntPos[j]+m_selfCheckPosture[1,j];
END_FOR
m_slefCheckPlanner[1].init(startJntPos,endJntPos,m_selfCheckMaxjntVel, m_selfCheckMaxjntAcc,m_selfCheckMaxjntJerk);

// other segments
IF m_selfCheckMotionNum>= 2 THEN
	FOR i:=2 TO m_selfCheckMotionNum DO 
		FOR j:=1 TO 7 DO 
			startJntPos[j]:=baseJntPos[j]+m_selfCheckPosture[i-1,j];
			endJntPos[j]:=baseJntPos[j]+m_selfCheckPosture[i,j];
		END_FOR
		m_slefCheckPlanner[i].init(startJntPos,endJntPos,m_selfCheckMaxjntVel, m_selfCheckMaxjntAcc,m_selfCheckMaxjntJerk);
	END_FOR
END_IF;

// update commands to arm
copyCmds(r_slaveArmCtrlCmd);
END_METHOD

END_FUNCTION_BLOCK

// ---- FBs_SlaveControllers/FB_SlaveCtrlMountInstru.TcPOU
// Brief: Mounting Instrument
FUNCTION_BLOCK PUBLIC FB_SlaveCtrlMountInstru EXTENDS FB_SlaveArmCtrlBase
VAR
	// mount status
	m_instruMountStatus :INT := 0;
	m_scopeMountStatus :INT := 0;
	m_ultrasoundMountStatus :INT :=0 ;
	
	// flag if joint is mounted
	m_jointMounted :ARRAY[1..5] OF BOOL := [5(FALSE)];
	
	// instrument mount motion range
	m_mountMotionAng :Vec5d :=[5(pi)];
	
	// instrument mount direction
	m_mountDir :Vec5i :=[1, 1, 1, 1, 1];
	
	// mount motion planning
	m_jntOTG :ARRAY[1..5] OF FB_secOrdTrajFilter;
	m_instruMountVel :LREAL := 4*PI;
	m_instruMountAcc :LREAL := 8*PI;
	
	//Joint 4 half-range angle of instrument
	m_instruJnt4HalfRangeAng :LREAL := 323*g_deg2Rad;
	
	// joint current threshold which indicate panel is buckled with instrument
	m_maxJntCurrent :Vec5d := [150, 150, 150, 180, 180];
	
	// command mount motion
	m_targetMountPos :Vec8d;
	
	// instrument zero position
	m_instruZeroDeviation :Vec5d;
	
	//ultrasound knife Reduce the current rotation Angle  J3
	m_ultraKnifeRotaAngleJ3 :LREAL := 30*g_deg2Rad;
	
	// ultrasound knife rotate angle zero position
	m_ultraKnifeRotAngZeroPos :LREAL := 4.50567;
	
	// joint position error
	m_jntPosErr :Vec5d;
	
	// endoscope motion angle to original position
	m_scopeJnt4CenterMotionAng :LREAL :=175*g_deg2Rad;
	m_scopeJnt5CenterMotionAng :LREAL :=150*g_deg2Rad;
	
	//instrument clamp error Id
	m_instruClampErrId : UINT;
	m_instruClampTime : LREAL;
	m_noCurrentTime : LREAL :=3;
	m_notReturnToZero : LREAL :=5;
END_VAR

// override this function in each exact controller
METHOD PROTECTED calcCmdJntPos : BOOL
VAR_IN_OUT CONSTANT
	i_endoscopePose : ST_Frame;
	i_masterStatus :ST_MasterStatus;
	i_setupStatus: ST_SetupStatus;
	i_slaveArm :FB_SlaveArm;
END_VAR

VAR 
END_VAR
// return directly if instrument/endoscope is not readed
IF i_slaveArm.instrument.onChipData.m_Error OR m_instruClampErrId >0  THEN
	return;
END_IF

IF i_slaveArm.instrument.onChipData.m_InstruReadSucceed AND InstruType_endoscope = i_slaveArm.instrument.m_instruType THEN
	mountEndoscope(i_slaveArm);
ELSIF i_slaveArm.instrument.onChipData.m_InstruReadSucceed AND (InstruType_UltrasoundKnifeS = i_slaveArm.instrument.m_instruType OR InstruType_UltrasoundKnifeU = i_slaveArm.instrument.m_instruType) THEN
	mountUltraKnife(i_slaveArm);
ELSE
	mountInstrument(i_slaveArm);
END_IF
m_instruClampErrId := instruClampStatus(i_slaveArm);
END_METHOD

METHOD PUBLIC init : BOOL
VAR_IN_OUT CONSTANT
	i_slaveArm	:FB_SlaveArm;
END_VAR
VAR_IN_OUT 
	r_slaveArmCtrlCmd :ST_SlaveArmCtrlCmds;
END_VAR

VAR
	i : INT;
END_VAR
// check if to hold the command joint position unchanged
m_holdLastCmds := checkToHoldLastCmds(i_slaveArm);

SUPER^.Init(i_slaveArm,r_slaveArmCtrlCmd);
m_jntOPMode[4] := DriverOPMode_PosTrq;
m_jntOPMode[5] := DriverOPMode_PosTrq;
m_jntOPMode[6] := DriverOPMode_PosTrq;
m_jntOPMode[7] := DriverOPMode_PosTrq;
m_jntOPMode[8] := DriverOPMode_PosTrq;

FOR i:=1 TO 5 DO
	m_targetMountPos[i+3]:=m_cmdJntPos[i+3];
	m_jntOTG[i].init(m_targetMountPos[i+3], 0,m_instruMountVel, m_instruMountAcc, g_slaveArmCtrlCycleTime);
	m_jointMounted[i]:=FALSE;
END_FOR

m_instruMountStatus:=0;
m_scopeMountStatus:=0;
m_ultrasoundMountStatus:=0;
m_instruClampErrId := 0;
m_instruClampTime := 0;
// update commands to arm
copyCmds(r_slaveArmCtrlCmd);
END_METHOD

PROPERTY instruClampErrId :  UINT
GET
instruClampErrId := m_instruClampErrId;
END_GET
END_PROPERTY

METHOD instruClampStatus : UINT
VAR_IN_OUT CONSTANT
	i_slaveArm :FB_SlaveArm;
END_VAR
//m_instruClampErrId=1 instrumen clamp the current does not reach the set value
//m_instruClampErrId=2 instrumen clamp position does not return to zero
m_instruClampTime := LIMIT(0,m_instruClampTime + g_slaveArmCtrlCycleTime,10);
IF i_slaveArm.instrument.onChipData.m_InstruReadSucceed THEN
	IF InstruType_endoscope = i_slaveArm.instrument.m_instruType THEN
		IF (m_scopeMountStatus=0 OR m_scopeMountStatus=1) AND m_instruClampTime>=m_noCurrentTime  THEN
			instruClampStatus := 1;
		ELSIF m_scopeMountStatus=3 AND m_instruClampTime>=m_notReturnToZero  THEN
			instruClampStatus := 2;
		END_IF
		
	ELSIF (InstruType_UltrasoundKnifeS = i_slaveArm.instrument.m_instruType OR InstruType_UltrasoundKnifeU = i_slaveArm.instrument.m_instruType) THEN
		IF (m_ultrasoundMountStatus=0) AND m_instruClampTime>=m_noCurrentTime  THEN
			instruClampStatus := 1;
		ELSIF (m_scopeMountStatus=3) AND m_instruClampTime>=m_notReturnToZero  THEN
			instruClampStatus := 2;
		END_IF
			
	ELSE
		IF (m_instruMountStatus=0) AND m_instruClampTime>=m_noCurrentTime  THEN
			instruClampStatus := 1;
		ELSIF (m_instruMountStatus=3) AND m_instruClampTime>=m_notReturnToZero  THEN
			instruClampStatus := 2;
		END_IF
	END_IF
END_IF
END_METHOD

METHOD mountEndoscope : BOOL
VAR_IN_OUT CONSTANT
	i_slaveArm :FB_SlaveArm;
END_VAR

VAR 
	i :INT;
	curJntPos :Vec8d;
END_VAR
curJntPos := i_slaveArm.curJntPos;

CASE m_scopeMountStatus OF
	//fix scope lock joint(joint 7)
	0:
		// other joints stay still
		FOR i:=1 TO 3 DO
			m_jointMounted[i] := TRUE;
			m_targetMountPos[i+3]:=curJntPos[i+3];
			m_jntOTG[i].init(m_targetMountPos[i+3], 0,m_instruMountVel, m_instruMountAcc, g_slaveArmCtrlCycleTime);
		END_FOR
	
		// check if buckled
		m_jointMounted[4]:=FALSE; 
		m_jointMounted[5]:=FALSE; 
		IF ABS(i_slaveArm.filtJntCurrent[7])> m_maxJntCurrent[4] THEN 
			m_jointMounted[4]:=TRUE;
			m_targetMountPos[7]:=curJntPos[7];
			m_jntOTG[4].init(m_targetMountPos[7], 0,m_instruMountVel, m_instruMountAcc, g_slaveArmCtrlCycleTime);
			m_scopeMountStatus:=1;
		ELSE
			m_targetMountPos[7]:=curJntPos[7]+m_mountMotionAng[4];
		END_IF

	1: // buckle scope rotate joint (joint 8)
		m_jointMounted[5]:=FALSE; 
		IF ABS(i_slaveArm.filtJntCurrent[8])> m_maxJntCurrent[5] THEN 
			m_jointMounted[5]:=TRUE;
			m_targetMountPos[8]:=curJntPos[8];
			m_jntOTG[5].init(m_targetMountPos[8], 0,m_instruMountVel, m_instruMountAcc, g_slaveArmCtrlCycleTime);
			m_scopeMountStatus:=2;
		ELSE
			m_targetMountPos[8]:=curJntPos[8]+m_mountMotionAng[5];
		END_IF
	

	2:// move back to zero position
		m_targetMountPos[7]:= curJntPos[7]-m_scopeJnt4CenterMotionAng;
		m_targetMountPos[8]:= curJntPos[8]-m_scopeJnt5CenterMotionAng;
		m_scopeMountStatus :=3;
		
		
	3:
		IF ABS(m_targetMountPos[7]-curJntPos[7]) <GVL_SlaveControlParameters.g_jntCtrlAngTolHigh AND 
				ABS(m_targetMountPos[8]-curJntPos[8]) <GVL_SlaveControlParameters.g_jntCtrlAngTolHigh THEN
			// record current joint position as offset for instrument
			i_slaveArm.instrument.initInstruJntPos(i_slaveArm.curJntPos);
			m_isFinished := TRUE;
		END_IF
		
END_CASE

// traj plan
FOR i:=1 TO 5 DO
	m_jntOTG[i].run(m_targetMountPos[i+3],0.0, o_cmdAcc=>m_cmdJntAcc[3+i],o_cmdVel=>m_cmdJntVel[3+i],o_cmdPos=>m_cmdJntPos[i+3]);
END_FOR
END_METHOD

METHOD mountInstrument : BOOL
VAR_IN_OUT CONSTANT
	i_slaveArm :FB_SlaveArm;
END_VAR

VAR 
	i :INT;
	curJntPos :Vec8d;
END_VAR
curJntPos := i_slaveArm.curJntPos;

// joint4 stay still if instrument has only on finger
IF i_slaveArm.instrument.m_isSingleFinger THEN
	m_jointMounted[1]:=TRUE;
END_IF

CASE m_instruMountStatus OF
	// To lock panel with instrument
	0:
		//buckle panel with instrument
		FOR i:=1 TO 4 DO
			// check if buckled 
			IF ABS(i_slaveArm.filtJntCurrent[i+3])> m_maxJntCurrent[i] THEN 
				m_jointMounted[i]:=TRUE;
				m_targetMountPos[i+3]:=curJntPos[i+3];
				m_jntOTG[i].init(m_targetMountPos[i+3], 0,m_instruMountVel, m_instruMountAcc, g_slaveArmCtrlCycleTime);
			END_IF
			
			// set target joint position
			IF FALSE = m_jointMounted[i] THEN
				IF i = 4 THEN
					m_targetMountPos[i+3]:=curJntPos[i+3]+m_mountMotionAng[i];
				ELSE
					m_targetMountPos[i+3]:=curJntPos[i+3]-m_mountMotionAng[i];
				END_IF
				
			END_IF
		END_FOR
		
		
		// check transition condition
		IF (m_jointMounted[1] AND m_jointMounted[2] AND m_jointMounted[3] AND m_jointMounted[4])  THEN
			IF i_slaveArm.instrument.onChipData.m_InstruReadSucceed THEN//Check whether the data is read successfully
				m_instruMountStatus:=1;
			END_IF
		END_IF
	
	1:// calculation deviates from the instrument zero position
		FOR i:=1 TO 4 DO
			m_instruZeroDeviation[i] :=  i_slaveArm.linkSingle[i+3] - i_slaveArm.instrument.onChipData.m_InstruPos[i];
		END_FOR
		m_instruMountStatus :=2;
	
	
	2:// move back to zero position
		FOR i:=1 TO 3 DO//J1-3
			IF m_instruZeroDeviation[i]>pi THEN
				m_instruZeroDeviation[i] := m_instruZeroDeviation[i] - 2*PI;
			ELSIF m_instruZeroDeviation[i]<-pi THEN
				m_instruZeroDeviation[i] := m_instruZeroDeviation[i] + 2*PI;
			END_IF
		END_FOR
		
		//joint4
		IF m_instruZeroDeviation[4]>0 AND m_instruZeroDeviation[4] < pi THEN
			m_instruZeroDeviation[4] := m_instruZeroDeviation[4] - 2*pi;
		ELSIF m_instruZeroDeviation[4]<0 AND m_instruZeroDeviation[4] > -pi THEN
			m_instruZeroDeviation[4] := m_instruZeroDeviation[4] + 2*pi;
		END_IF
		
		// set target joint position
		FOR i:=1 TO 4 DO
			m_targetMountPos[i+3]:=curJntPos[i+3] - m_instruZeroDeviation[i];
		END_FOR
		m_instruMountStatus :=3;
	
	3: // make fingers is closed
		//m_instruMountStatus :=4;
		FOR i:=1 TO 4 DO 
			m_jointMounted[i]:=FALSE;
			m_jntPosErr[i]:=m_targetMountPos[i+3]-curJntPos[i+3];
			IF ABS(m_jntPosErr[i]) <GVL_SlaveControlParameters.g_jntCtrlAngTolLow OR 
					ABS( i_slaveArm.linkSingle[i+3] - i_slaveArm.instrument.onChipData.m_InstruPos[i]) <5*g_deg2rad THEN
				m_jointMounted[i]:=TRUE;
				//EXIT;
			END_IF
		END_FOR
		
		IF ABS(i_slaveArm.filtJntCurrent[7])> m_maxJntCurrent[4] AND ABS(i_slaveArm.curJntVel[7])< 1*g_deg2rad AND
				ABS( i_slaveArm.linkSingle[7] - i_slaveArm.instrument.onChipData.m_InstruPos[4]) >10*g_deg2rad AND NOT m_jointMounted[4] THEN 
			m_instruZeroDeviation[4] :=  i_slaveArm.linkSingle[7] - i_slaveArm.instrument.onChipData.m_InstruPos[4];
			m_jointMounted[4]:=TRUE;
			IF m_instruZeroDeviation[4]>=0 AND m_instruZeroDeviation[4] < pi THEN
				m_instruZeroDeviation[4] := m_instruZeroDeviation[4] - 2*pi;
			ELSIF m_instruZeroDeviation[4]<0 AND m_instruZeroDeviation[4] > -pi THEN
				m_instruZeroDeviation[4] := m_instruZeroDeviation[4] + 2*pi;	
			END_IF
		ELSE
			m_instruZeroDeviation[4] := 0;
		END_IF
		
		IF (m_jointMounted[1] AND m_jointMounted[2] AND m_jointMounted[3] AND m_jointMounted[4])  THEN
			m_instruMountStatus :=4;
		END_IF
		
		IF m_instruMountStatus =4 AND NOT( i_slaveArm.instrument.m_isSingleFinger) THEN
			m_targetMountPos[4] := curJntPos[4]+g_gripperCloseAng;
			m_targetMountPos[5] := curJntPos[5]+g_gripperCloseAng;
			m_targetMountPos[7] := curJntPos[7]-m_instruZeroDeviation[4];
		END_IF
		
	4:
		m_isFinished :=  ABS(m_targetMountPos[4]-curJntPos[4]) < GVL_SlaveControlParameters.g_jntCtrlAngTolLow AND
			 ABS(m_targetMountPos[5]-curJntPos[5]) < GVL_SlaveControlParameters.g_jntCtrlAngTolLow AND ABS(m_targetMountPos[7]-curJntPos[7]) < GVL_SlaveControlParameters.g_jntCtrlAngTolLow;
			 
		// record current joint position as offset for instrument
		i_slaveArm.instrument.initInstruJntPos(i_slaveArm.curJntPos);

END_CASE

// traj plan
FOR i:=1 TO 4 DO
	m_jntOTG[i].run(m_targetMountPos[i+3],0.0, o_cmdAcc=>m_cmdJntAcc[3+i],o_cmdVel=>m_cmdJntVel[3+i],o_cmdPos=>m_cmdJntPos[i+3]);
END_FOR
END_METHOD

METHOD mountUltraKnife : BOOL
VAR_IN_OUT CONSTANT
	i_slaveArm :FB_SlaveArm;
END_VAR

VAR 
	i :INT;
	curJntPos :Vec8d;
END_VAR
curJntPos := i_slaveArm.curJntPos;

m_jointMounted[1]:=TRUE;
m_jointMounted[2]:=TRUE;


CASE m_ultrasoundMountStatus OF 
	// To lock panel with instrument
	0:
		//buckle panel with instrument
		FOR i:=3 TO 5 DO
			// check if buckled 
			IF ABS(i_slaveArm.filtJntCurrent[i+3])> m_maxJntCurrent[i] THEN 
				m_jointMounted[i]:=TRUE;
				m_targetMountPos[i+3]:=curJntPos[i+3];
				m_jntOTG[i].init(m_targetMountPos[i+3], 0,m_instruMountVel, m_instruMountAcc, g_slaveArmCtrlCycleTime);
			END_IF
			
			// set target joint position
			IF FALSE = m_jointMounted[i] THEN
				IF i = 5 THEN
					m_targetMountPos[i+3]:=curJntPos[i+3]+m_mountMotionAng[i];
				ELSE
					m_targetMountPos[i+3]:=curJntPos[i+3]-m_mountMotionAng[i];
				END_IF
				
			END_IF
		END_FOR

		// check transition condition
		IF ( m_jointMounted[3] AND m_jointMounted[4] AND m_jointMounted[5] )  THEN
			IF i_slaveArm.instrument.onChipData.m_InstruReadSucceed THEN//Check whether the data is read successfully
				m_ultrasoundMountStatus:=1;
			END_IF
		END_IF

	1:
		//m_jntOPMode[8] := DriverOPMode_Trq;
		// calculation deviates from the instrument zero position
		m_instruZeroDeviation[3] :=  m_ultraKnifeRotaAngleJ3;
		m_instruZeroDeviation[4] :=  i_slaveArm.linkSingle[7] - m_ultraKnifeRotAngZeroPos;
		m_ultrasoundMountStatus :=2;
		
	2:// move back to zero position
		//joint4
		IF m_instruZeroDeviation[4]>0 AND m_instruZeroDeviation[4] < pi THEN
			m_instruZeroDeviation[4] := m_instruZeroDeviation[4] - 2*pi;
		ELSIF m_instruZeroDeviation[4]<0 AND m_instruZeroDeviation[4] > -pi THEN
			m_instruZeroDeviation[4] := m_instruZeroDeviation[4] + 2*pi;
		END_IF
	
		// set target joint position
		m_targetMountPos[6]:=curJntPos[6] + m_instruZeroDeviation[3];
		m_targetMountPos[7]:=curJntPos[7] - m_instruZeroDeviation[4];
		m_targetMountPos[8]:=curJntPos[8] - m_instruZeroDeviation[4];

		m_ultrasoundMountStatus :=3;

	3:
		// joint8 in passive mode
		m_jntOPMode[8] := DriverOPMode_Trq;
		
		m_isFinished:=TRUE;
		FOR i:=3 TO 4 DO 
			m_jntPosErr[i]:=m_targetMountPos[i+3]-curJntPos[i+3];
			IF ABS(m_jntPosErr[i]) >GVL_SlaveControlParameters.g_jntCtrlAngTolLow  THEN
				m_isFinished := FALSE;
				EXIT;
			END_IF
		END_FOR	
		
		// record current joint position as offset for instrument
		i_slaveArm.instrument.initInstruJntPos(i_slaveArm.curJntPos);

END_CASE


// traj plan
FOR i:=1 TO 5 DO
	m_jntOTG[i].run(m_targetMountPos[i+3],0.0, o_cmdAcc=>m_cmdJntAcc[3+i],o_cmdVel=>m_cmdJntVel[3+i],o_cmdPos=>m_cmdJntPos[i+3]);
END_FOR
END_METHOD

END_FUNCTION_BLOCK

